KUKA KRL program: EPS_2_251825_SA24_A_20260116064100.src

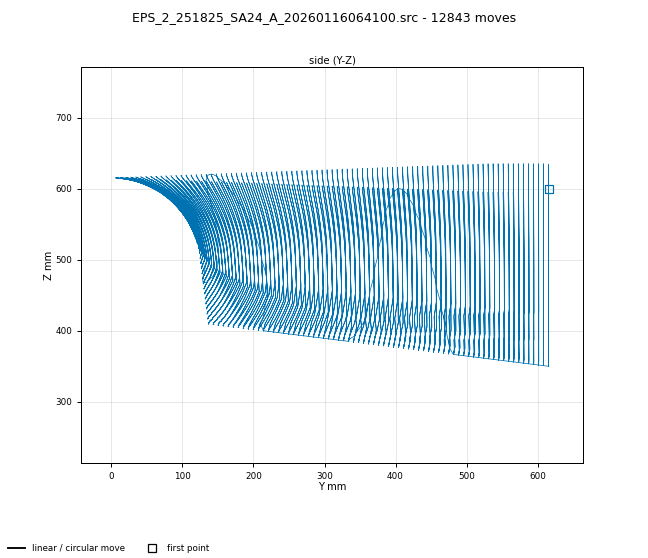
[picture p0: tool path of EPS_2_251825_SA24_A_20260116064100.src, 12843 of 12845 moves have a stored position in this frame; points joined in program order, loops and branches not executed]
&ACCESS RVP
&REL 4
&COMMENT QRS 19112012
&PARAM EDITMASK = *
DEF PART()
EXT BAS (BAS_COMMAND :IN,REAL :IN )
INT I
BAS (#INITMOV,0 )

;KUKA QRS Post kuka4.cps  Date:22-06-2017 !

File_ID=2983

QRS_PRE_INIT()

;Init var - Until changes are made in qrs_pre_init
Outlet_Square_prg=0
Inlet_1_Square_prg=0
Inlet_2_Square_prg=0
Inlet_3_Square_prg=0
Inlet_4_Square_prg=0
Inlet_5_Square_prg=0

Outlet_1={X 0.000, Y 530.070, Z 534.500, B 0.000, E1 0.000 }
Inlet_1={X 0.000, Y 532.930, Z 494.500, B 0.000, E1 180.000 }
Outlet_1_type=201
Inlet_1_type=201
;QRS#1=Sidecore dimensions
;QRS#2=200-8" PVC SDR 35
;QRS#3=200-8" PVC SDR 35
;QRS#4=
;QRS#5=
;QRS#6=
;QRS#7=
;QRS#8=
;QRS#9=12-08 PSX
;QRS#10=12-08 PSX
;QRS#11=
;QRS#12=
;QRS#13=
;QRS#14=
;QRS#15=
;QRS#16=1220x127x914 3'
;QRS#17=EPS Height
;QRS#18=635
;QRS#19=*
;QRS#20= UPDATED VERSION 22-06-2017
;QRS#21=*
Outlet_Square=0100
Inlet_1_Square=0100
Inlet_2_Square=0
Inlet_3_Square=0
Inlet_4_Square=0
Inlet_5_Square=0
Mill_Square=1
Outlet_Square_Prg=204
Inlet_1_Square_prg=204

QRS_INIT()

$ADVANCE=5

; T1
PTP {E1 173.589,E2 173.589}
PTP {X 0,Y 615.513,A -85,B 0,C 180,E1 173.589,E2 173.589,E3 0,E4 0,E5 0,E6 0}
QRS_SPEED_INIT()
LIN {X 0,Y 615.513,Z 600,A -85,B 0,C 180,E1 173.589,E2 173.589,E3 0,E4 0,E5 0,E6 0} C_VEL
LIN {X 0,Y 615.513,Z 359.866,A -85,B 0,C 180,E1 173.589,E2 173.589} C_VEL
LIN {X 0,Y 615.513,Z 351.692,A -85,B 0,C 180,E1 173.589,E2 173.589} C_VEL
LIN {X 0,Y 615.497,Z 349.692,A -85,B 0,C 180,E1 173.403,E2 173.403} C_VEL
LIN {X 0,Y 615.488,Z 349.69,A -85,B 0,C 180,E1 170.801,E2 170.801} C_VEL
LIN {X 0,Y 615.478,Z 349.685,A -85,B 0,C 180,E1 168.139,E2 168.139} C_VEL
LIN {X 0,Y 615.497,Z 349.694,A -85,B 0,C 180,E1 165.451,E2 165.451} C_VEL
LIN {X 0,Y 615.493,Z 349.685,A -85,B 0,C 180,E1 162.73,E2 162.73} C_VEL
LIN {X 0,Y 615.479,Z 349.687,A -85,B 0,C 180,E1 159.967,E2 159.967} C_VEL
LIN {X 0,Y 615.488,Z 349.695,A -85,B 0,C 180,E1 157.155,E2 157.155} C_VEL
LIN {X 0,Y 615.484,Z 349.683,A -85,B 0,C 180,E1 154.429,E2 154.429} C_VEL
LIN {X 0,Y 615.497,Z 349.697,A -85,B 0,C 180,E1 151.546,E2 151.546} C_VEL
LIN {X 0,Y 615.487,Z 349.686,A -85,B 0,C 180,E1 148.912,E2 148.912} C_VEL
LIN {X 0,Y 615.484,Z 349.683,A -85,B 0,C 180,E1 146.464,E2 146.464} C_VEL
LIN {X 0,Y 615.488,Z 349.702,A -85,B 0,C 180,E1 143.575,E2 143.575} C_VEL
LIN {X 0,Y 615.481,Z 349.686,A -85,B 0,C 180,E1 140.937,E2 140.937} C_VEL
LIN {X 0,Y 615.485,Z 349.683,A -85,B 0,C 180,E1 138.526,E2 138.526} C_VEL
LIN {X 0,Y 615.491,Z 349.695,A -85,B 0,C 180,E1 135.85,E2 135.85} C_VEL
LIN {X 0,Y 615.483,Z 349.686,A -85,B 0,C 180,E1 133.047,E2 133.047} C_VEL
LIN {X 0,Y 615.482,Z 349.684,A -85,B 0,C 180,E1 130.606,E2 130.606} C_VEL
LIN {X 0,Y 615.484,Z 349.695,A -85,B 0,C 180,E1 128.011,E2 128.011} C_VEL
LIN {X 0,Y 615.486,Z 349.696,A -85,B 0,C 180,E1 125.615,E2 125.615} C_VEL
LIN {X 0,Y 615.477,Z 349.688,A -85,B 0,C 180,E1 123.236,E2 123.236} C_VEL
LIN {X 0,Y 615.492,Z 349.681,A -85,B 0,C 180,E1 120.919,E2 120.919} C_VEL
LIN {X 0,Y 615.477,Z 349.689,A -85,B 0,C 180,E1 118.448,E2 118.448} C_VEL
LIN {X 0,Y 615.489,Z 349.695,A -85,B 0,C 180,E1 115.715,E2 115.715} C_VEL
LIN {X 0,Y 615.486,Z 349.683,A -85,B 0,C 180,E1 112.844,E2 112.844} C_VEL
LIN {X 0,Y 615.485,Z 349.703,A -85,B 0,C 180,E1 110.032,E2 110.032} C_VEL
LIN {X 0,Y 615.481,Z 349.809,A -85,B 0,C 180,E1 108.602,E2 108.602} C_VEL
LIN {X 0,Y 615.486,Z 366.721,A -85,B 0,C 180,E1 105.735,E2 105.735} C_VEL
LIN {X 0,Y 615.497,Z 384.117,A -85,B 0,C 180,E1 102.823,E2 102.823} C_VEL
LIN {X 0,Y 615.478,Z 491.809,A -85,B 0,C 180,E1 101.527,E2 101.527} C_VEL
LIN {X 0,Y 615.481,Z 504.75,A -85,B 0,C 180,E1 101.235,E2 101.235} C_VEL
LIN {X 0,Y 615.493,Z 516.589,A -85,B 0,C 180,E1 100.843,E2 100.843} C_VEL
LIN {X 0,Y 615.485,Z 527.572,A -85,B 0,C 180,E1 100.36,E2 100.36} C_VEL
LIN {X 0,Y 615.492,Z 539.308,A -85,B 0,C 180,E1 99.696,E2 99.696} C_VEL
LIN {X 0,Y 615.499,Z 549.77,A -85,B 0,C 180,E1 98.95,E2 98.95} C_VEL
LIN {X 0,Y 615.498,Z 558.332,A -85,B 0,C 180,E1 98.206,E2 98.206} C_VEL
LIN {X 0,Y 615.497,Z 566.211,A -85,B 0,C 180,E1 97.38,E2 97.38} C_VEL
LIN {X 0,Y 615.497,Z 573.9,A -85,B 0,C 180,E1 96.392,E2 96.392} C_VEL
LIN {X 0,Y 615.497,Z 580.959,A -85,B 0,C 180,E1 95.241,E2 95.241} C_VEL
LIN {X 0,Y 615.494,Z 585.658,A -85,B 0,C 180,E1 94.256,E2 94.256} C_VEL
LIN {X 0,Y 615.494,Z 589.255,A -85,B 0,C 180,E1 93.273,E2 93.273} C_VEL
LIN {X 0,Y 615.496,Z 591.115,A -85,B 0,C 180,E1 92.618,E2 92.618} C_VEL
LIN {X 0,Y 615.499,Z 592.533,A -85,B 0,C 180,E1 91.963,E2 91.963} C_VEL
LIN {X 0,Y 615.496,Z 594.142,A -85,B 0,C 180,E1 90.654,E2 90.654} C_VEL
LIN {X 0,Y 615.495,Z 594.384,A -85,B 0,C 180,E1 90,E2 90} C_VEL
LIN {X 0,Y 615.495,Z 594.206,A -85,B 0,C 180,E1 89.346,E2 89.346} C_VEL
LIN {X 0,Y 615.499,Z 592.682,A -85,B 0,C 180,E1 88.037,E2 88.037} C_VEL
LIN {X 0,Y 615.498,Z 591.341,A -85,B 0,C 180,E1 87.382,E2 87.382} C_VEL
LIN {X 0,Y 615.496,Z 588.494,A -85,B 0,C 180,E1 86.399,E2 86.399} C_VEL
LIN {X 0,Y 615.499,Z 584.635,A -85,B 0,C 180,E1 85.416,E2 85.416} C_VEL
LIN {X 0,Y 615.498,Z 579.652,A -85,B 0,C 180,E1 84.43,E2 84.43} C_VEL
LIN {X 0,Y 615.496,Z 573.208,A -85,B 0,C 180,E1 83.418,E2 83.418} C_VEL
LIN {X 0,Y 615.497,Z 565.538,A -85,B 0,C 180,E1 82.455,E2 82.455} C_VEL
LIN {X 0,Y 615.498,Z 555.761,A -85,B 0,C 180,E1 81.464,E2 81.464} C_VEL
LIN {X 0,Y 615.498,Z 545.496,A -85,B 0,C 180,E1 80.636,E2 80.636} C_VEL
LIN {X 0,Y 615.488,Z 533.934,A -85,B 0,C 180,E1 79.889,E2 79.889} C_VEL
LIN {X 0,Y 615.495,Z 522.053,A -85,B 0,C 180,E1 79.292,E2 79.292} C_VEL
LIN {X 0,Y 615.483,Z 509.169,A -85,B 0,C 180,E1 78.807,E2 78.807} C_VEL
LIN {X 0,Y 615.476,Z 496.573,A -85,B 0,C 180,E1 78.473,E2 78.473} C_VEL
LIN {X 0,Y 615.48,Z 483.461,A -85,B 0,C 180,E1 78.265,E2 78.265} C_VEL
LIN {X 0,Y 615.499,Z 384.153,A -85,B 0,C 180,E1 77.093,E2 77.093} C_VEL
LIN {X 0,Y 615.486,Z 367.257,A -85,B 0,C 180,E1 74.265,E2 74.265} C_VEL
LIN {X 0,Y 615.487,Z 350.325,A -85,B 0,C 180,E1 71.396,E2 71.396} C_VEL
LIN {X 0,Y 615.491,Z 349.685,A -85,B 0,C 180,E1 71.268,E2 71.268} C_VEL
LIN {X 0,Y 615.477,Z 349.687,A -85,B 0,C 180,E1 68.568,E2 68.568} C_VEL
LIN {X 0,Y 615.482,Z 349.696,A -85,B 0,C 180,E1 65.728,E2 65.728} C_VEL
LIN {X 0,Y 615.486,Z 349.683,A -85,B 0,C 180,E1 62.956,E2 62.956} C_VEL
LIN {X 0,Y 615.497,Z 349.695,A -85,B 0,C 180,E1 60.204,E2 60.204} C_VEL
LIN {X 0,Y 615.48,Z 349.688,A -85,B 0,C 180,E1 57.543,E2 57.543} C_VEL
LIN {X 0,Y 615.499,Z 349.68,A -85,B 0,C 180,E1 55.187,E2 55.187} C_VEL
LIN {X 0,Y 615.477,Z 349.688,A -85,B 0,C 180,E1 52.758,E2 52.758} C_VEL
LIN {X 0,Y 615.48,Z 349.695,A -85,B 0,C 180,E1 49.912,E2 49.912} C_VEL
LIN {X 0,Y 615.475,Z 349.689,A -85,B 0,C 180,E1 47.647,E2 47.647} C_VEL
LIN {X 0,Y 615.48,Z 349.686,A -85,B 0,C 180,E1 44.932,E2 44.932} C_VEL
LIN {X 0,Y 615.486,Z 349.695,A -85,B 0,C 180,E1 42.082,E2 42.082} C_VEL
LIN {X 0,Y 615.477,Z 349.688,A -85,B 0,C 180,E1 39.751,E2 39.751} C_VEL
LIN {X 0,Y 615.478,Z 349.688,A -85,B 0,C 180,E1 36.937,E2 36.937} C_VEL
LIN {X 0,Y 615.481,Z 349.692,A -85,B 0,C 180,E1 34.023,E2 34.023} C_VEL
LIN {X 0,Y 615.479,Z 349.686,A -85,B 0,C 180,E1 31.686,E2 31.686} C_VEL
LIN {X 0,Y 615.486,Z 349.683,A -85,B 0,C 180,E1 29.407,E2 29.407} C_VEL
LIN {X 0,Y 615.495,Z 349.698,A -85,B 0,C 180,E1 26.444,E2 26.444} C_VEL
LIN {X 0,Y 615.486,Z 349.683,A -85,B 0,C 180,E1 23.557,E2 23.557} C_VEL
LIN {X 0,Y 615.486,Z 349.698,A -85,B 0,C 180,E1 20.731,E2 20.731} C_VEL
LIN {X 0,Y 615.477,Z 349.687,A -85,B 0,C 180,E1 17.957,E2 17.957} C_VEL
LIN {X 0,Y 615.491,Z 349.686,A -85,B 0,C 180,E1 15.226,E2 15.226} C_VEL
LIN {X 0,Y 615.493,Z 349.695,A -85,B 0,C 180,E1 12.53,E2 12.53} C_VEL
LIN {X 0,Y 615.477,Z 349.685,A -85,B 0,C 180,E1 9.862,E2 9.862} C_VEL
LIN {X 0,Y 615.49,Z 349.689,A -85,B 0,C 180,E1 7.216,E2 7.216} C_VEL
LIN {X 0,Y 615.494,Z 349.693,A -85,B 0,C 180,E1 4.585,E2 4.585} C_VEL
LIN {X 0,Y 615.477,Z 349.685,A -85,B 0,C 180,E1 1.963,E2 1.963} C_VEL
LIN {X 0,Y 615.489,Z 349.688,A -85,B 0,C 180,E1 -0.654,E2 -0.654} C_VEL
LIN {X 0,Y 615.496,Z 349.693,A -85,B 0,C 180,E1 -3.273,E2 -3.273} C_VEL
LIN {X 0,Y 615.476,Z 349.685,A -85,B 0,C 180,E1 -5.899,E2 -5.899} C_VEL
LIN {X 0,Y 615.491,Z 349.688,A -85,B 0,C 180,E1 -8.537,E2 -8.537} C_VEL
LIN {X 0,Y 615.494,Z 349.692,A -85,B 0,C 180,E1 -11.193,E2 -11.193} C_VEL
LIN {X 0,Y 615.474,Z 349.685,A -85,B 0,C 180,E1 -13.933,E2 -13.933} C_VEL
LIN {X 0,Y 615.493,Z 349.692,A -85,B 0,C 180,E1 -16.587,E2 -16.587} C_VEL
LIN {X 0,Y 615.49,Z 349.687,A -85,B 0,C 180,E1 -19.338,E2 -19.338} C_VEL
LIN {X 0,Y 615.479,Z 349.687,A -85,B 0,C 180,E1 -22.137,E2 -22.137} C_VEL
LIN {X 0,Y 615.488,Z 349.694,A -85,B 0,C 180,E1 -24.992,E2 -24.992} C_VEL
LIN {X 0,Y 615.487,Z 349.688,A -85,B 0,C 180,E1 -27.177,E2 -27.177} C_VEL
LIN {X 0,Y 615.477,Z 349.685,A -85,B 0,C 180,E1 -29.795,E2 -29.795} C_VEL
LIN {X 0,Y 615.495,Z 349.694,A -85,B 0,C 180,E1 -32.457,E2 -32.457} C_VEL
LIN {X 0,Y 615.49,Z 349.695,A -85,B 0,C 180,E1 -34.815,E2 -34.815} C_VEL
LIN {X 0,Y 615.491,Z 349.684,A -85,B 0,C 180,E1 -37.242,E2 -37.242} C_VEL
LIN {X 0,Y 615.484,Z 349.69,A -85,B 0,C 180,E1 -40.09,E2 -40.09} C_VEL
LIN {X 0,Y 615.499,Z 349.695,A -85,B 0,C 180,E1 -42.352,E2 -42.352} C_VEL
LIN {X 0,Y 615.484,Z 349.686,A -85,B 0,C 180,E1 -45.069,E2 -45.069} C_VEL
LIN {X 0,Y 615.477,Z 349.69,A -85,B 0,C 180,E1 -47.921,E2 -47.921} C_VEL
LIN {X 0,Y 615.497,Z 349.696,A -85,B 0,C 180,E1 -50.252,E2 -50.252} C_VEL
LIN {X 0,Y 615.485,Z 349.685,A -85,B 0,C 180,E1 -53.064,E2 -53.064} C_VEL
LIN {X 0,Y 615.491,Z 349.681,A -85,B 0,C 180,E1 -55.299,E2 -55.299} C_VEL
LIN {X 0,Y 615.477,Z 349.688,A -85,B 0,C 180,E1 -57.671,E2 -57.671} C_VEL
LIN {X 0,Y 615.499,Z 349.699,A -85,B 0,C 180,E1 -60.204,E2 -60.204} C_VEL
LIN {X 0,Y 615.487,Z 349.684,A -85,B 0,C 180,E1 -62.956,E2 -62.956} C_VEL
LIN {X 0,Y 615.478,Z 349.691,A -85,B 0,C 180,E1 -65.728,E2 -65.728} C_VEL
LIN {X 0,Y 615.48,Z 349.76,A -85,B 0,C 180,E1 -67.438,E2 -67.438} C_VEL
LIN {X 0,Y 615.494,Z 369.694,A -85,B 0,C 180,E1 -70.142,E2 -70.142} C_VEL
LIN {X 0,Y 615.493,Z 391.661,A -85,B 0,C 180,E1 -73.072,E2 -73.072} C_VEL
LIN {X 0,Y 615.498,Z 414.417,A -85,B 0,C 180,E1 -76.064,E2 -76.064} C_VEL
LIN {X 0,Y 615.497,Z 422.467,A -85,B 0,C 180,E1 -77.114,E2 -77.114} C_VEL
LIN {X 0,Y 615.479,Z 530.847,A -85,B 0,C 180,E1 -78.411,E2 -78.411} C_VEL
LIN {X 0,Y 615.478,Z 543.355,A -85,B 0,C 180,E1 -78.682,E2 -78.682} C_VEL
LIN {X 0,Y 615.491,Z 556.569,A -85,B 0,C 180,E1 -79.111,E2 -79.111} C_VEL
LIN {X 0,Y 615.478,Z 568.483,A -85,B 0,C 180,E1 -79.639,E2 -79.639} C_VEL
LIN {X 0,Y 615.487,Z 579.999,A -85,B 0,C 180,E1 -80.304,E2 -80.304} C_VEL
LIN {X 0,Y 615.499,Z 590.344,A -85,B 0,C 180,E1 -81.05,E2 -81.05} C_VEL
LIN {X 0,Y 615.497,Z 598.814,A -85,B 0,C 180,E1 -81.794,E2 -81.794} C_VEL
LIN {X 0,Y 615.498,Z 606.608,A -85,B 0,C 180,E1 -82.62,E2 -82.62} C_VEL
LIN {X 0,Y 615.496,Z 614.204,A -85,B 0,C 180,E1 -83.608,E2 -83.608} C_VEL
LIN {X 0,Y 615.498,Z 621.205,A -85,B 0,C 180,E1 -84.759,E2 -84.759} C_VEL
LIN {X 0,Y 615.493,Z 625.852,A -85,B 0,C 180,E1 -85.744,E2 -85.744} C_VEL
LIN {X 0,Y 615.495,Z 629.399,A -85,B 0,C 180,E1 -86.727,E2 -86.727} C_VEL
LIN {X 0,Y 615.497,Z 631.233,A -85,B 0,C 180,E1 -87.382,E2 -87.382} C_VEL
LIN {X 0,Y 615.497,Z 632.608,A -85,B 0,C 180,E1 -88.037,E2 -88.037} C_VEL
LIN {X 0,Y 615.496,Z 634.174,A -85,B 0,C 180,E1 -89.346,E2 -89.346} C_VEL
LIN {X 0,Y 615.494,Z 634.389,A -85,B 0,C 180,E1 -90,E2 -90} C_VEL
LIN {X 0,Y 615.496,Z 633.58,A -85,B 0,C 180,E1 -91.309,E2 -91.309} C_VEL
LIN {X 0,Y 615.497,Z 632.608,A -85,B 0,C 180,E1 -91.963,E2 -91.963} C_VEL
LIN {X 0,Y 615.497,Z 631.233,A -85,B 0,C 180,E1 -92.618,E2 -92.618} C_VEL
LIN {X 0,Y 615.496,Z 628.35,A -85,B 0,C 180,E1 -93.601,E2 -93.601} C_VEL
LIN {X 0,Y 615.498,Z 624.442,A -85,B 0,C 180,E1 -94.584,E2 -94.584} C_VEL
LIN {X 0,Y 615.499,Z 619.406,A -85,B 0,C 180,E1 -95.57,E2 -95.57} C_VEL
LIN {X 0,Y 615.497,Z 612.869,A -85,B 0,C 180,E1 -96.583,E2 -96.583} C_VEL
LIN {X 0,Y 615.497,Z 605.135,A -85,B 0,C 180,E1 -97.545,E2 -97.545} C_VEL
LIN {X 0,Y 615.498,Z 597.047,A -85,B 0,C 180,E1 -98.371,E2 -98.371} C_VEL
LIN {X 0,Y 615.499,Z 587.17,A -85,B 0,C 180,E1 -99.198,E2 -99.198} C_VEL
LIN {X 0,Y 615.488,Z 575.985,A -85,B 0,C 180,E1 -99.945,E2 -99.945} C_VEL
LIN {X 0,Y 615.481,Z 565.029,A -85,B 0,C 180,E1 -100.527,E2 -100.527} C_VEL
LIN {X 0,Y 615.49,Z 552.453,A -85,B 0,C 180,E1 -101.041,E2 -101.041} C_VEL
LIN {X 0,Y 615.477,Z 540.079,A -85,B 0,C 180,E1 -101.401,E2 -101.401} C_VEL
LIN {X 0,Y 615.481,Z 526.487,A -85,B 0,C 180,E1 -101.652,E2 -101.652} C_VEL
LIN {X 0,Y 615.497,Z 422.467,A -85,B 0,C 180,E1 -102.886,E2 -102.886} C_VEL
LIN {X 0,Y 615.49,Z 399.409,A -85,B 0,C 180,E1 -105.905,E2 -105.905} C_VEL
LIN {X 0,Y 615.494,Z 377.451,A -85,B 0,C 180,E1 -108.818,E2 -108.818} C_VEL
LIN {X 0,Y 615.483,Z 356.76,A -85,B 0,C 180,E1 -111.607,E2 -111.607} C_VEL
LIN {X 0,Y 615.481,Z 349.685,A -85,B 0,C 180,E1 -112.593,E2 -112.593} C_VEL
LIN {X 0,Y 615.488,Z 349.683,A -85,B 0,C 180,E1 -114.991,E2 -114.991} C_VEL
LIN {X 0,Y 615.487,Z 349.698,A -85,B 0,C 180,E1 -117.914,E2 -117.914} C_VEL
LIN {X 0,Y 615.476,Z 349.692,A -85,B 0,C 180,E1 -120.16,E2 -120.16} C_VEL
LIN {X 0,Y 615.479,Z 349.686,A -85,B 0,C 180,E1 -122.457,E2 -122.457} C_VEL
LIN {X 0,Y 615.499,Z 349.68,A -85,B 0,C 180,E1 -124.813,E2 -124.813} C_VEL
LIN {X 0,Y 615.483,Z 349.69,A -85,B 0,C 180,E1 -127.241,E2 -127.241} C_VEL
LIN {X 0,Y 615.477,Z 349.691,A -85,B 0,C 180,E1 -130.088,E2 -130.088} C_VEL
LIN {X 0,Y 615.475,Z 349.686,A -85,B 0,C 180,E1 -132.353,E2 -132.353} C_VEL
LIN {X 0,Y 615.486,Z 349.688,A -85,B 0,C 180,E1 -135.067,E2 -135.067} C_VEL
LIN {X 0,Y 615.486,Z 349.69,A -85,B 0,C 180,E1 -137.918,E2 -137.918} C_VEL
LIN {X 0,Y 615.477,Z 349.686,A -85,B 0,C 180,E1 -140.249,E2 -140.249} C_VEL
LIN {X 0,Y 615.488,Z 349.69,A -85,B 0,C 180,E1 -143.062,E2 -143.062} C_VEL
LIN {X 0,Y 615.481,Z 349.688,A -85,B 0,C 180,E1 -145.978,E2 -145.978} C_VEL
LIN {X 0,Y 615.476,Z 349.685,A -85,B 0,C 180,E1 -148.314,E2 -148.314} C_VEL
LIN {X 0,Y 615.488,Z 349.684,A -85,B 0,C 180,E1 -150.594,E2 -150.594} C_VEL
LIN {X 0,Y 615.497,Z 349.691,A -85,B 0,C 180,E1 -153.556,E2 -153.556} C_VEL
LIN {X 0,Y 615.486,Z 349.683,A -85,B 0,C 180,E1 -156.444,E2 -156.444} C_VEL
LIN {X 0,Y 615.497,Z 349.699,A -85,B 0,C 180,E1 -159.27,E2 -159.27} C_VEL
LIN {X 0,Y 615.477,Z 349.685,A -85,B 0,C 180,E1 -162.043,E2 -162.043} C_VEL
LIN {X 0,Y 615.492,Z 349.69,A -85,B 0,C 180,E1 -164.774,E2 -164.774} C_VEL
LIN {X 0,Y 615.491,Z 349.69,A -85,B 0,C 180,E1 -167.47,E2 -167.47} C_VEL
LIN {X 0,Y 615.477,Z 349.685,A -85,B 0,C 180,E1 -170.138,E2 -170.138} C_VEL
LIN {X 0,Y 615.494,Z 349.692,A -85,B 0,C 180,E1 -172.784,E2 -172.784} C_VEL
LIN {X 0,Y 615.492,Z 349.689,A -85,B 0,C 180,E1 -175.415,E2 -175.415} C_VEL
LIN {X 0,Y 615.477,Z 349.685,A -85,B 0,C 180,E1 -178.037,E2 -178.037} C_VEL
LIN {X 0,Y 615.494,Z 349.692,A -85,B 0,C 180,E1 -180.654,E2 -180.654} C_VEL
LIN {X 0,Y 615.492,Z 349.689,A -85,B 0,C 180,E1 -183.273,E2 -183.273} C_VEL
LIN {X 0,Y 615.476,Z 349.685,A -85,B 0,C 180,E1 -185.899,E2 -185.899} C_VEL
LIN {X 0,Y 615.497,Z 349.692,A -85,B 0,C 180,E1 -186.597,E2 -186.597} C_VEL
LIN {X 0,Y 614.817,Z 349.838,A -85,B 0,C 180,E1 -187.143,E2 -187.143} C_VEL
LIN {X 0,Y 611.977,Z 350.249,A -85,B 0,C 180,E1 -188.029,E2 -188.029} C_VEL
LIN {X 0,Y 609.583,Z 350.561,A -85,B 0,C 180,E1 -188.741,E2 -188.741} C_VEL
LIN {X 0,Y 608.546,Z 350.679,A -85,B 0,C 180,E1 -189.291,E2 -189.291} C_VEL
LIN {X 0,Y 608.456,Z 350.688,A -85,B 0,C 180,E1 -189.477,E2 -189.477} C_VEL
LIN {X 0,Y 608.456,Z 350.687,A -85,B 0,C 180,E1 -192,E2 -192} C_VEL
LIN {X 0,Y 608.481,Z 350.694,A -85,B 0,C 180,E1 -194.72,E2 -194.72} C_VEL
LIN {X 0,Y 608.453,Z 350.688,A -85,B 0,C 180,E1 -197.477,E2 -197.477} C_VEL
LIN {X 0,Y 608.462,Z 350.69,A -85,B 0,C 180,E1 -200.274,E2 -200.274} C_VEL
LIN {X 0,Y 608.486,Z 350.691,A -85,B 0,C 180,E1 -202.485,E2 -202.485} C_VEL
LIN {X 0,Y 608.449,Z 350.689,A -85,B 0,C 180,E1 -205.301,E2 -205.301} C_VEL
LIN {X 0,Y 608.444,Z 350.688,A -85,B 0,C 180,E1 -207.518,E2 -207.518} C_VEL
LIN {X 0,Y 608.46,Z 350.688,A -85,B 0,C 180,E1 -209.973,E2 -209.973} C_VEL
LIN {X 0,Y 608.467,Z 350.696,A -85,B 0,C 180,E1 -212.525,E2 -212.525} C_VEL
LIN {X 0,Y 608.436,Z 350.69,A -85,B 0,C 180,E1 -215.278,E2 -215.278} C_VEL
LIN {X 0,Y 608.467,Z 350.687,A -85,B 0,C 180,E1 -217.747,E2 -217.747} C_VEL
LIN {X 0,Y 608.449,Z 350.698,A -85,B 0,C 180,E1 -220.33,E2 -220.33} C_VEL
LIN {X 0,Y 608.483,Z 350.684,A -85,B 0,C 180,E1 -223.312,E2 -223.312} C_VEL
LIN {X 0,Y 608.467,Z 350.693,A -85,B 0,C 180,E1 -226.132,E2 -226.132} C_VEL
LIN {X 0,Y 608.451,Z 350.69,A -85,B 0,C 180,E1 -228.824,E2 -228.824} C_VEL
LIN {X 0,Y 608.468,Z 350.686,A -85,B 0,C 180,E1 -231.413,E2 -231.413} C_VEL
LIN {X 0,Y 608.476,Z 350.691,A -85,B 0,C 180,E1 -233.951,E2 -233.951} C_VEL
LIN {X 0,Y 608.448,Z 350.696,A -85,B 0,C 180,E1 -236.329,E2 -236.329} C_VEL
LIN {X 0,Y 608.476,Z 350.686,A -85,B 0,C 180,E1 -238.728,E2 -238.728} C_VEL
LIN {X 0,Y 608.469,Z 350.686,A -85,B 0,C 180,E1 -241.381,E2 -241.381} C_VEL
LIN {X 0,Y 608.471,Z 350.692,A -85,B 0,C 180,E1 -244.28,E2 -244.28} C_VEL
LIN {X 0,Y 608.449,Z 350.688,A -85,B 0,C 180,E1 -246.877,E2 -246.877} C_VEL
LIN {X 0,Y 608.459,Z 350.693,A -85,B 0,C 180,E1 -249.726,E2 -249.726} C_VEL
LIN {X 0,Y 608.467,Z 350.778,A -85,B 0,C 180,E1 -251.331,E2 -251.331} C_VEL
LIN {X 0,Y 608.497,Z 366.845,A -85,B 0,C 180,E1 -254.08,E2 -254.08} C_VEL
LIN {X 0,Y 608.485,Z 384.321,A -85,B 0,C 180,E1 -257.027,E2 -257.027} C_VEL
LIN {X 0,Y 608.573,Z 393.682,A -85,B 0,C 180,E1 -257.156,E2 -257.156} C_VEL
LIN {X 0,Y 608.545,Z 490.809,A -85,B 0,C 180,E1 -258.319,E2 -258.319} C_VEL
LIN {X 0,Y 608.524,Z 504.124,A -85,B 0,C 180,E1 -258.614,E2 -258.614} C_VEL
LIN {X 0,Y 608.527,Z 517.379,A -85,B 0,C 180,E1 -259.056,E2 -259.056} C_VEL
LIN {X 0,Y 608.495,Z 529.373,A -85,B 0,C 180,E1 -259.603,E2 -259.603} C_VEL
LIN {X 0,Y 608.505,Z 540.793,A -85,B 0,C 180,E1 -260.276,E2 -260.276} C_VEL
LIN {X 0,Y 608.474,Z 551.086,A -85,B 0,C 180,E1 -261.03,E2 -261.03} C_VEL
LIN {X 0,Y 608.464,Z 560.352,A -85,B 0,C 180,E1 -261.866,E2 -261.866} C_VEL
LIN {X 0,Y 608.466,Z 569.325,A -85,B 0,C 180,E1 -262.868,E2 -262.868} C_VEL
LIN {X 0,Y 608.444,Z 576.556,A -85,B 0,C 180,E1 -263.867,E2 -263.867} C_VEL
LIN {X 0,Y 608.462,Z 581.435,A -85,B 0,C 180,E1 -264.698,E2 -264.698} C_VEL
LIN {X 0,Y 608.439,Z 586.179,A -85,B 0,C 180,E1 -265.694,E2 -265.694} C_VEL
LIN {X 0,Y 608.425,Z 589.812,A -85,B 0,C 180,E1 -266.689,E2 -266.689} C_VEL
LIN {X 0,Y 608.425,Z 591.691,A -85,B 0,C 180,E1 -267.352,E2 -267.352} C_VEL
LIN {X 0,Y 608.444,Z 593.127,A -85,B 0,C 180,E1 -268.014,E2 -268.014} C_VEL
LIN {X 0,Y 608.439,Z 594.752,A -85,B 0,C 180,E1 -269.338,E2 -269.338} C_VEL
LIN {X 0,Y 608.435,Z 594.995,A -85,B 0,C 180,E1 -270,E2 -270} C_VEL
LIN {X 0,Y 608.438,Z 594.815,A -85,B 0,C 180,E1 -270.662,E2 -270.662} C_VEL
LIN {X 0,Y 608.444,Z 593.276,A -85,B 0,C 180,E1 -271.986,E2 -271.986} C_VEL
LIN {X 0,Y 608.426,Z 591.919,A -85,B 0,C 180,E1 -272.648,E2 -272.648} C_VEL
LIN {X 0,Y 608.449,Z 589.042,A -85,B 0,C 180,E1 -273.642,E2 -273.642} C_VEL
LIN {X 0,Y 608.433,Z 585.143,A -85,B 0,C 180,E1 -274.638,E2 -274.638} C_VEL
LIN {X 0,Y 608.45,Z 580.113,A -85,B 0,C 180,E1 -275.634,E2 -275.634} C_VEL
LIN {X 0,Y 608.441,Z 573.796,A -85,B 0,C 180,E1 -276.633,E2 -276.633} C_VEL
LIN {X 0,Y 608.475,Z 565.88,A -85,B 0,C 180,E1 -277.633,E2 -277.633} C_VEL
LIN {X 0,Y 608.472,Z 556.038,A -85,B 0,C 180,E1 -278.636,E2 -278.636} C_VEL
LIN {X 0,Y 608.48,Z 545.717,A -85,B 0,C 180,E1 -279.473,E2 -279.473} C_VEL
LIN {X 0,Y 608.485,Z 534.104,A -85,B 0,C 180,E1 -280.229,E2 -280.229} C_VEL
LIN {X 0,Y 608.526,Z 522.887,A -85,B 0,C 180,E1 -280.802,E2 -280.802} C_VEL
LIN {X 0,Y 608.523,Z 510.37,A -85,B 0,C 180,E1 -281.287,E2 -281.287} C_VEL
LIN {X 0,Y 608.521,Z 497.571,A -85,B 0,C 180,E1 -281.639,E2 -281.639} C_VEL
LIN {X 0,Y 608.534,Z 485.31,A -85,B 0,C 180,E1 -281.85,E2 -281.85} C_VEL
LIN {X 0,Y 608.463,Z 384.352,A -85,B 0,C 180,E1 -283.059,E2 -283.059} C_VEL
LIN {X 0,Y 608.497,Z 367.375,A -85,B 0,C 180,E1 -285.92,E2 -285.92} C_VEL
LIN {X 0,Y 608.471,Z 350.687,A -85,B 0,C 180,E1 -288.775,E2 -288.775} C_VEL
LIN {X 0,Y 608.467,Z 350.69,A -85,B 0,C 180,E1 -291.691,E2 -291.691} C_VEL
LIN {X 0,Y 608.452,Z 350.69,A -85,B 0,C 180,E1 -294.57,E2 -294.57} C_VEL
LIN {X 0,Y 608.476,Z 350.685,A -85,B 0,C 180,E1 -297.206,E2 -297.206} C_VEL
LIN {X 0,Y 608.47,Z 350.696,A -85,B 0,C 180,E1 -299.971,E2 -299.971} C_VEL
LIN {X 0,Y 608.456,Z 350.689,A -85,B 0,C 180,E1 -302.521,E2 -302.521} C_VEL
LIN {X 0,Y 608.447,Z 350.69,A -85,B 0,C 180,E1 -305.276,E2 -305.276} C_VEL
LIN {X 0,Y 608.466,Z 350.695,A -85,B 0,C 180,E1 -307.745,E2 -307.745} C_VEL
LIN {X 0,Y 608.446,Z 350.691,A -85,B 0,C 180,E1 -310.328,E2 -310.328} C_VEL
LIN {X 0,Y 608.447,Z 350.688,A -85,B 0,C 180,E1 -312.959,E2 -312.959} C_VEL
LIN {X 0,Y 608.458,Z 350.698,A -85,B 0,C 180,E1 -315.735,E2 -315.735} C_VEL
LIN {X 0,Y 608.459,Z 350.686,A -85,B 0,C 180,E1 -318.657,E2 -318.657} C_VEL
LIN {X 0,Y 608.464,Z 350.692,A -85,B 0,C 180,E1 -321.411,E2 -321.411} C_VEL
LIN {X 0,Y 608.471,Z 350.69,A -85,B 0,C 180,E1 -323.95,E2 -323.95} C_VEL
LIN {X 0,Y 608.461,Z 350.687,A -85,B 0,C 180,E1 -326.329,E2 -326.329} C_VEL
LIN {X 0,Y 608.472,Z 350.685,A -85,B 0,C 180,E1 -328.726,E2 -328.726} C_VEL
LIN {X 0,Y 608.475,Z 350.693,A -85,B 0,C 180,E1 -331.377,E2 -331.377} C_VEL
LIN {X 0,Y 608.464,Z 350.686,A -85,B 0,C 180,E1 -334.278,E2 -334.278} C_VEL
LIN {X 0,Y 608.449,Z 350.69,A -85,B 0,C 180,E1 -336.876,E2 -336.876} C_VEL
LIN {X 0,Y 608.469,Z 350.695,A -85,B 0,C 180,E1 -339.318,E2 -339.318} C_VEL
LIN {X 0,Y 608.446,Z 350.691,A -85,B 0,C 180,E1 -341.828,E2 -341.828} C_VEL
LIN {X 0,Y 608.47,Z 350.686,A -85,B 0,C 180,E1 -344.594,E2 -344.594} C_VEL
LIN {X 0,Y 608.48,Z 350.694,A -85,B 0,C 180,E1 -347.323,E2 -347.323} C_VEL
LIN {X 0,Y 608.451,Z 350.688,A -85,B 0,C 180,E1 -350.023,E2 -350.023} C_VEL
LIN {X 0,Y 608.481,Z 350.686,A -85,B 0,C 180,E1 -352.701,E2 -352.701} C_VEL
LIN {X 0,Y 608.462,Z 350.693,A -85,B 0,C 180,E1 -355.362,E2 -355.362} C_VEL
LIN {X 0,Y 608.448,Z 350.688,A -85,B 0,C 180,E1 -358.014,E2 -358.014} C_VEL
LIN {X 0,Y 608.482,Z 350.687,A -85,B 0,C 180,E1 -360.662,E2 -360.662} C_VEL
LIN {X 0,Y 608.486,Z 350.689,A -85,B 0,C 180,E1 -363.311,E2 -363.311} C_VEL
LIN {X 0,Y 608.452,Z 350.687,A -85,B 0,C 180,E1 -365.967,E2 -365.967} C_VEL
LIN {X 0,Y 608.46,Z 350.691,A -85,B 0,C 180,E1 -368.636,E2 -368.636} C_VEL
LIN {X 0,Y 608.477,Z 350.689,A -85,B 0,C 180,E1 -371.324,E2 -371.324} C_VEL
LIN {X 0,Y 608.458,Z 350.687,A -85,B 0,C 180,E1 -374.038,E2 -374.038} C_VEL
LIN {X 0,Y 608.477,Z 350.694,A -85,B 0,C 180,E1 -376.783,E2 -376.783} C_VEL
LIN {X 0,Y 608.451,Z 350.688,A -85,B 0,C 180,E1 -379.571,E2 -379.571} C_VEL
LIN {X 0,Y 608.485,Z 350.689,A -85,B 0,C 180,E1 -382.485,E2 -382.485} C_VEL
LIN {X 0,Y 608.45,Z 350.69,A -85,B 0,C 180,E1 -385.301,E2 -385.301} C_VEL
LIN {X 0,Y 608.445,Z 350.689,A -85,B 0,C 180,E1 -387.518,E2 -387.518} C_VEL
LIN {X 0,Y 608.46,Z 350.687,A -85,B 0,C 180,E1 -389.973,E2 -389.973} C_VEL
LIN {X 0,Y 608.467,Z 350.694,A -85,B 0,C 180,E1 -392.525,E2 -392.525} C_VEL
LIN {X 0,Y 608.441,Z 350.69,A -85,B 0,C 180,E1 -395.278,E2 -395.278} C_VEL
LIN {X 0,Y 608.468,Z 350.686,A -85,B 0,C 180,E1 -397.747,E2 -397.747} C_VEL
LIN {X 0,Y 608.476,Z 350.692,A -85,B 0,C 180,E1 -400.333,E2 -400.333} C_VEL
LIN {X 0,Y 608.483,Z 350.684,A -85,B 0,C 180,E1 -403.312,E2 -403.312} C_VEL
LIN {X 0,Y 608.468,Z 350.691,A -85,B 0,C 180,E1 -406.132,E2 -406.132} C_VEL
LIN {X 0,Y 608.456,Z 350.691,A -85,B 0,C 180,E1 -408.825,E2 -408.825} C_VEL
LIN {X 0,Y 608.469,Z 350.685,A -85,B 0,C 180,E1 -411.413,E2 -411.413} C_VEL
LIN {X 0,Y 608.477,Z 350.689,A -85,B 0,C 180,E1 -413.951,E2 -413.951} C_VEL
LIN {X 0,Y 608.464,Z 350.696,A -85,B 0,C 180,E1 -416.33,E2 -416.33} C_VEL
LIN {X 0,Y 608.477,Z 350.687,A -85,B 0,C 180,E1 -418.728,E2 -418.728} C_VEL
LIN {X 0,Y 608.469,Z 350.686,A -85,B 0,C 180,E1 -421.381,E2 -421.381} C_VEL
LIN {X 0,Y 608.474,Z 350.694,A -85,B 0,C 180,E1 -424.279,E2 -424.279} C_VEL
LIN {X 0,Y 608.45,Z 350.69,A -85,B 0,C 180,E1 -426.877,E2 -426.877} C_VEL
LIN {X 0,Y 608.503,Z 350.824,A -85,B 0,C 180,E1 -427.312,E2 -427.312} C_VEL
LIN {X 0,Y 608.567,Z 369.705,A -85,B 0,C 180,E1 -429.906,E2 -429.906} C_VEL
LIN {X 0,Y 608.521,Z 391.71,A -85,B 0,C 180,E1 -432.872,E2 -432.872} C_VEL
LIN {X 0,Y 608.476,Z 413.716,A -85,B 0,C 180,E1 -435.792,E2 -435.792} C_VEL
LIN {X 0,Y 608.504,Z 422.696,A -85,B 0,C 180,E1 -436.974,E2 -436.974} C_VEL
LIN {X 0,Y 608.538,Z 530.962,A -85,B 0,C 180,E1 -438.277,E2 -438.277} C_VEL
LIN {X 0,Y 608.514,Z 544.226,A -85,B 0,C 180,E1 -438.572,E2 -438.572} C_VEL
LIN {X 0,Y 608.517,Z 556.599,A -85,B 0,C 180,E1 -438.981,E2 -438.981} C_VEL
LIN {X 0,Y 608.498,Z 568.639,A -85,B 0,C 180,E1 -439.519,E2 -439.519} C_VEL
LIN {X 0,Y 608.48,Z 580.201,A -85,B 0,C 180,E1 -440.191,E2 -440.191} C_VEL
LIN {X 0,Y 608.485,Z 590.596,A -85,B 0,C 180,E1 -440.946,E2 -440.946} C_VEL
LIN {X 0,Y 608.475,Z 599.114,A -85,B 0,C 180,E1 -441.699,E2 -441.699} C_VEL
LIN {X 0,Y 608.471,Z 606.962,A -85,B 0,C 180,E1 -442.534,E2 -442.534} C_VEL
LIN {X 0,Y 608.461,Z 614.287,A -85,B 0,C 180,E1 -443.485,E2 -443.485} C_VEL
LIN {X 0,Y 608.45,Z 619.867,A -85,B 0,C 180,E1 -444.366,E2 -444.366} C_VEL
LIN {X 0,Y 608.432,Z 624.951,A -85,B 0,C 180,E1 -445.362,E2 -445.362} C_VEL
LIN {X 0,Y 608.449,Z 628.896,A -85,B 0,C 180,E1 -446.358,E2 -446.358} C_VEL
LIN {X 0,Y 608.425,Z 631.809,A -85,B 0,C 180,E1 -447.352,E2 -447.352} C_VEL
LIN {X 0,Y 608.442,Z 633.201,A -85,B 0,C 180,E1 -448.014,E2 -448.014} C_VEL
LIN {X 0,Y 608.438,Z 634.783,A -85,B 0,C 180,E1 -449.338,E2 -449.338} C_VEL
LIN {X 0,Y 608.434,Z 635,A -85,B 0,C 180,E1 -450,E2 -450} C_VEL
LIN {X 0,Y 608.448,Z 634.184,A -85,B 0,C 180,E1 -451.324,E2 -451.324} C_VEL
LIN {X 0,Y 608.442,Z 633.201,A -85,B 0,C 180,E1 -451.986,E2 -451.986} C_VEL
LIN {X 0,Y 608.425,Z 631.809,A -85,B 0,C 180,E1 -452.648,E2 -452.648} C_VEL
LIN {X 0,Y 608.449,Z 628.896,A -85,B 0,C 180,E1 -453.642,E2 -453.642} C_VEL
LIN {X 0,Y 608.432,Z 624.95,A -85,B 0,C 180,E1 -454.638,E2 -454.638} C_VEL
LIN {X 0,Y 608.437,Z 618.877,A -85,B 0,C 180,E1 -455.801,E2 -455.801} C_VEL
LIN {X 0,Y 608.462,Z 612.236,A -85,B 0,C 180,E1 -456.799,E2 -456.799} C_VEL
LIN {X 0,Y 608.455,Z 603.991,A -85,B 0,C 180,E1 -457.8,E2 -457.8} C_VEL
LIN {X 0,Y 608.472,Z 595.538,A -85,B 0,C 180,E1 -458.636,E2 -458.636} C_VEL
LIN {X 0,Y 608.471,Z 585.094,A -85,B 0,C 180,E1 -459.473,E2 -459.473} C_VEL
LIN {X 0,Y 608.494,Z 574.76,A -85,B 0,C 180,E1 -460.144,E2 -460.144} C_VEL
LIN {X 0,Y 608.521,Z 563.256,A -85,B 0,C 180,E1 -460.74,E2 -460.74} C_VEL
LIN {X 0,Y 608.531,Z 550.887,A -85,B 0,C 180,E1 -461.225,E2 -461.225} C_VEL
LIN {X 0,Y 608.537,Z 537.45,A -85,B 0,C 180,E1 -461.597,E2 -461.597} C_VEL
LIN {X 0,Y 608.546,Z 525.105,A -85,B 0,C 180,E1 -461.808,E2 -461.808} C_VEL
LIN {X 0,Y 608.493,Z 422.615,A -85,B 0,C 180,E1 -463.037,E2 -463.037} C_VEL
LIN {X 0,Y 608.497,Z 400.771,A -85,B 0,C 180,E1 -465.92,E2 -465.92} C_VEL
LIN {X 0,Y 608.517,Z 379.797,A -85,B 0,C 180,E1 -468.728,E2 -468.728} C_VEL
LIN {X 0,Y 608.557,Z 360.644,A -85,B 0,C 180,E1 -471.332,E2 -471.332} C_VEL
LIN {X 0,Y 608.457,Z 350.689,A -85,B 0,C 180,E1 -472.714,E2 -472.714} C_VEL
LIN {X 0,Y 608.45,Z 350.69,A -85,B 0,C 180,E1 -475.3,E2 -475.3} C_VEL
LIN {X 0,Y 608.449,Z 350.694,A -85,B 0,C 180,E1 -477.517,E2 -477.517} C_VEL
LIN {X 0,Y 608.472,Z 350.692,A -85,B 0,C 180,E1 -479.972,E2 -479.972} C_VEL
LIN {X 0,Y 608.455,Z 350.687,A -85,B 0,C 180,E1 -482.521,E2 -482.521} C_VEL
LIN {X 0,Y 608.454,Z 350.691,A -85,B 0,C 180,E1 -485.276,E2 -485.276} C_VEL
LIN {X 0,Y 608.467,Z 350.695,A -85,B 0,C 180,E1 -487.745,E2 -487.745} C_VEL
LIN {X 0,Y 608.445,Z 350.689,A -85,B 0,C 180,E1 -490.328,E2 -490.328} C_VEL
LIN {X 0,Y 608.473,Z 350.691,A -85,B 0,C 180,E1 -493.309,E2 -493.309} C_VEL
LIN {X 0,Y 608.468,Z 350.687,A -85,B 0,C 180,E1 -496.13,E2 -496.13} C_VEL
LIN {X 0,Y 608.455,Z 350.688,A -85,B 0,C 180,E1 -498.823,E2 -498.823} C_VEL
LIN {X 0,Y 608.468,Z 350.695,A -85,B 0,C 180,E1 -501.412,E2 -501.412} C_VEL
LIN {X 0,Y 608.471,Z 350.688,A -85,B 0,C 180,E1 -503.95,E2 -503.95} C_VEL
LIN {X 0,Y 608.461,Z 350.686,A -85,B 0,C 180,E1 -506.329,E2 -506.329} C_VEL
LIN {X 0,Y 608.473,Z 350.686,A -85,B 0,C 180,E1 -508.726,E2 -508.726} C_VEL
LIN {X 0,Y 608.478,Z 350.694,A -85,B 0,C 180,E1 -511.377,E2 -511.377} C_VEL
LIN {X 0,Y 608.446,Z 350.689,A -85,B 0,C 180,E1 -513.964,E2 -513.964} C_VEL
LIN {X 0,Y 608.46,Z 350.686,A -85,B 0,C 180,E1 -516.155,E2 -516.155} C_VEL
LIN {X 0,Y 608.47,Z 350.685,A -85,B 0,C 180,E1 -518.308,E2 -518.308} C_VEL
LIN {X 0,Y 608.472,Z 350.694,A -85,B 0,C 180,E1 -521.28,E2 -521.28} C_VEL
LIN {X 0,Y 608.457,Z 350.687,A -85,B 0,C 180,E1 -523.906,E2 -523.906} C_VEL
LIN {X 0,Y 608.466,Z 350.689,A -85,B 0,C 180,E1 -526.644,E2 -526.644} C_VEL
LIN {X 0,Y 608.473,Z 350.691,A -85,B 0,C 180,E1 -529.35,E2 -529.35} C_VEL
LIN {X 0,Y 608.47,Z 350.685,A -85,B 0,C 180,E1 -532.033,E2 -532.033} C_VEL
LIN {X 0,Y 608.471,Z 350.69,A -85,B 0,C 180,E1 -534.698,E2 -534.698} C_VEL
LIN {X 0,Y 608.484,Z 350.688,A -85,B 0,C 180,E1 -537.352,E2 -537.352} C_VEL
LIN {X 0,Y 608.468,Z 350.685,A -85,B 0,C 180,E1 -540,E2 -540} C_VEL
LIN {X 0,Y 608.486,Z 350.689,A -85,B 0,C 180,E1 -542.648,E2 -542.648} C_VEL
LIN {X 0,Y 608.469,Z 350.689,A -85,B 0,C 180,E1 -545.302,E2 -545.302} C_VEL
LIN {X 0,Y 608.471,Z 350.685,A -85,B 0,C 180,E1 -547.967,E2 -547.967} C_VEL
LIN {X 0,Y 608.456,Z 350.688,A -85,B 0,C 180,E1 -549.477,E2 -549.477} C_VEL
LIN {X 0,Y 607.774,Z 350.774,A -85,B 0,C 180,E1 -550.03,E2 -550.03} C_VEL
LIN {X 0,Y 604.916,Z 351.136,A -85,B 0,C 180,E1 -550.927,E2 -550.927} C_VEL
LIN {X 0,Y 602.515,Z 351.431,A -85,B 0,C 180,E1 -551.648,E2 -551.648} C_VEL
LIN {X 0,Y 601.489,Z 351.557,A -85,B 0,C 180,E1 -552.205,E2 -552.205} C_VEL
LIN {X 0,Y 601.408,Z 351.568,A -85,B 0,C 180,E1 -552.394,E2 -552.394} C_VEL
LIN {X 0,Y 601.432,Z 351.57,A -85,B 0,C 180,E1 -554.897,E2 -554.897} C_VEL
LIN {X 0,Y 601.432,Z 351.568,A -85,B 0,C 180,E1 -556.986,E2 -556.986} C_VEL
LIN {X 0,Y 601.404,Z 351.565,A -85,B 0,C 180,E1 -559.81,E2 -559.81} C_VEL
LIN {X 0,Y 601.448,Z 351.57,A -85,B 0,C 180,E1 -562.682,E2 -562.682} C_VEL
LIN {X 0,Y 601.401,Z 351.572,A -85,B 0,C 180,E1 -564.879,E2 -564.879} C_VEL
LIN {X 0,Y 601.419,Z 351.564,A -85,B 0,C 180,E1 -567.868,E2 -567.868} C_VEL
LIN {X 0,Y 601.42,Z 351.568,A -85,B 0,C 180,E1 -570.165,E2 -570.165} C_VEL
LIN {X 0,Y 601.426,Z 351.569,A -85,B 0,C 180,E1 -572.718,E2 -572.718} C_VEL
LIN {X 0,Y 601.391,Z 351.568,A -85,B 0,C 180,E1 -575.113,E2 -575.113} C_VEL
LIN {X 0,Y 601.43,Z 351.562,A -85,B 0,C 180,E1 -577.42,E2 -577.42} C_VEL
LIN {X 0,Y 601.406,Z 351.569,A -85,B 0,C 180,E1 -579.996,E2 -579.996} C_VEL
LIN {X 0,Y 601.434,Z 351.567,A -85,B 0,C 180,E1 -582.669,E2 -582.669} C_VEL
LIN {X 0,Y 601.422,Z 351.563,A -85,B 0,C 180,E1 -585.483,E2 -585.483} C_VEL
LIN {X 0,Y 601.42,Z 351.572,A -85,B 0,C 180,E1 -588.408,E2 -588.408} C_VEL
LIN {X 0,Y 601.434,Z 351.563,A -85,B 0,C 180,E1 -590.876,E2 -590.876} C_VEL
LIN {X 0,Y 601.441,Z 351.564,A -85,B 0,C 180,E1 -593.735,E2 -593.735} C_VEL
LIN {X 0,Y 601.431,Z 351.571,A -85,B 0,C 180,E1 -596.065,E2 -596.065} C_VEL
LIN {X 0,Y 601.429,Z 351.562,A -85,B 0,C 180,E1 -599.059,E2 -599.059} C_VEL
LIN {X 0,Y 601.429,Z 351.563,A -85,B 0,C 180,E1 -601.374,E2 -601.374} C_VEL
LIN {X 0,Y 601.401,Z 351.569,A -85,B 0,C 180,E1 -603.637,E2 -603.637} C_VEL
LIN {X 0,Y 601.453,Z 351.567,A -85,B 0,C 180,E1 -605.86,E2 -605.86} C_VEL
LIN {X 0,Y 601.405,Z 351.566,A -85,B 0,C 180,E1 -608.761,E2 -608.761} C_VEL
LIN {X 0,Y 601.462,Z 351.726,A -85,B 0,C 180,E1 -611.27,E2 -611.27} C_VEL
LIN {X 0,Y 601.487,Z 367.861,A -85,B 0,C 180,E1 -614.063,E2 -614.063} C_VEL
LIN {X 0,Y 601.413,Z 384.324,A -85,B 0,C 180,E1 -616.871,E2 -616.871} C_VEL
LIN {X 0,Y 601.68,Z 388.362,A -85,B 0,C 180,E1 -616.942,E2 -616.942} C_VEL
LIN {X 0,Y 601.615,Z 490.839,A -85,B 0,C 180,E1 -618.183,E2 -618.183} C_VEL
LIN {X 0,Y 601.562,Z 503.383,A -85,B 0,C 180,E1 -618.459,E2 -618.459} C_VEL
LIN {X 0,Y 601.541,Z 516.517,A -85,B 0,C 180,E1 -618.894,E2 -618.894} C_VEL
LIN {X 0,Y 601.517,Z 527.754,A -85,B 0,C 180,E1 -619.396,E2 -619.396} C_VEL
LIN {X 0,Y 601.485,Z 539.526,A -85,B 0,C 180,E1 -620.076,E2 -620.076} C_VEL
LIN {X 0,Y 601.444,Z 550.035,A -85,B 0,C 180,E1 -620.839,E2 -620.839} C_VEL
LIN {X 0,Y 601.429,Z 558.642,A -85,B 0,C 180,E1 -621.601,E2 -621.601} C_VEL
LIN {X 0,Y 601.418,Z 566.57,A -85,B 0,C 180,E1 -622.446,E2 -622.446} C_VEL
LIN {X 0,Y 601.376,Z 573.89,A -85,B 0,C 180,E1 -623.393,E2 -623.393} C_VEL
LIN {X 0,Y 601.372,Z 579.613,A -85,B 0,C 180,E1 -624.299,E2 -624.299} C_VEL
LIN {X 0,Y 601.336,Z 584.754,A -85,B 0,C 180,E1 -625.307,E2 -625.307} C_VEL
LIN {X 0,Y 601.367,Z 588.744,A -85,B 0,C 180,E1 -626.315,E2 -626.315} C_VEL
LIN {X 0,Y 601.324,Z 591.693,A -85,B 0,C 180,E1 -627.321,E2 -627.321} C_VEL
LIN {X 0,Y 601.343,Z 593.127,A -85,B 0,C 180,E1 -627.991,E2 -627.991} C_VEL
LIN {X 0,Y 601.339,Z 594.753,A -85,B 0,C 180,E1 -629.33,E2 -629.33} C_VEL
LIN {X 0,Y 601.336,Z 594.996,A -85,B 0,C 180,E1 -630,E2 -630} C_VEL
LIN {X 0,Y 601.339,Z 594.815,A -85,B 0,C 180,E1 -630.67,E2 -630.67} C_VEL
LIN {X 0,Y 601.343,Z 593.276,A -85,B 0,C 180,E1 -632.009,E2 -632.009} C_VEL
LIN {X 0,Y 601.326,Z 591.917,A -85,B 0,C 180,E1 -632.679,E2 -632.679} C_VEL
LIN {X 0,Y 601.368,Z 589.04,A -85,B 0,C 180,E1 -633.685,E2 -633.685} C_VEL
LIN {X 0,Y 601.337,Z 585.141,A -85,B 0,C 180,E1 -634.693,E2 -634.693} C_VEL
LIN {X 0,Y 601.373,Z 580.11,A -85,B 0,C 180,E1 -635.701,E2 -635.701} C_VEL
LIN {X 0,Y 601.382,Z 573.792,A -85,B 0,C 180,E1 -636.711,E2 -636.711} C_VEL
LIN {X 0,Y 601.396,Z 565.876,A -85,B 0,C 180,E1 -637.723,E2 -637.723} C_VEL
LIN {X 0,Y 601.436,Z 556.032,A -85,B 0,C 180,E1 -638.737,E2 -638.737} C_VEL
LIN {X 0,Y 601.45,Z 545.711,A -85,B 0,C 180,E1 -639.585,E2 -639.585} C_VEL
LIN {X 0,Y 601.487,Z 534.093,A -85,B 0,C 180,E1 -640.349,E2 -640.349} C_VEL
LIN {X 0,Y 601.549,Z 522.876,A -85,B 0,C 180,E1 -640.929,E2 -640.929} C_VEL
LIN {X 0,Y 601.55,Z 510.332,A -85,B 0,C 180,E1 -641.42,E2 -641.42} C_VEL
LIN {X 0,Y 601.587,Z 497.548,A -85,B 0,C 180,E1 -641.775,E2 -641.775} C_VEL
LIN {X 0,Y 601.601,Z 485.271,A -85,B 0,C 180,E1 -641.989,E2 -641.989} C_VEL
LIN {X 0,Y 601.52,Z 385.126,A -85,B 0,C 180,E1 -643.191,E2 -643.191} C_VEL
LIN {X 0,Y 601.421,Z 384.348,A -85,B 0,C 180,E1 -643.214,E2 -643.214} C_VEL
LIN {X 0,Y 601.472,Z 368.385,A -85,B 0,C 180,E1 -645.937,E2 -645.937} C_VEL
LIN {X 0,Y 601.509,Z 352.928,A -85,B 0,C 180,E1 -648.609,E2 -648.609} C_VEL
LIN {X 0,Y 601.427,Z 351.565,A -85,B 0,C 180,E1 -648.875,E2 -648.875} C_VEL
LIN {X 0,Y 601.408,Z 351.566,A -85,B 0,C 180,E1 -651.239,E2 -651.239} C_VEL
LIN {X 0,Y 601.462,Z 351.568,A -85,B 0,C 180,E1 -654.14,E2 -654.14} C_VEL
LIN {X 0,Y 601.448,Z 351.56,A -85,B 0,C 180,E1 -657.111,E2 -657.111} C_VEL
LIN {X 0,Y 601.423,Z 351.565,A -85,B 0,C 180,E1 -659.392,E2 -659.392} C_VEL
LIN {X 0,Y 601.412,Z 351.571,A -85,B 0,C 180,E1 -661.725,E2 -661.725} C_VEL
LIN {X 0,Y 601.429,Z 351.569,A -85,B 0,C 180,E1 -664.117,E2 -664.117} C_VEL
LIN {X 0,Y 601.411,Z 351.565,A -85,B 0,C 180,E1 -666.581,E2 -666.581} C_VEL
LIN {X 0,Y 601.44,Z 351.567,A -85,B 0,C 180,E1 -669.535,E2 -669.535} C_VEL
LIN {X 0,Y 601.406,Z 351.565,A -85,B 0,C 180,E1 -672.59,E2 -672.59} C_VEL
LIN {X 0,Y 601.421,Z 351.569,A -85,B 0,C 180,E1 -675.481,E2 -675.481} C_VEL
LIN {X 0,Y 601.422,Z 351.564,A -85,B 0,C 180,E1 -678.406,E2 -678.406} C_VEL
LIN {X 0,Y 601.43,Z 351.563,A -85,B 0,C 180,E1 -680.875,E2 -680.875} C_VEL
LIN {X 0,Y 601.437,Z 351.57,A -85,B 0,C 180,E1 -683.733,E2 -683.733} C_VEL
LIN {X 0,Y 601.426,Z 351.563,A -85,B 0,C 180,E1 -686.686,E2 -686.686} C_VEL
LIN {X 0,Y 601.426,Z 351.566,A -85,B 0,C 180,E1 -689.058,E2 -689.058} C_VEL
LIN {X 0,Y 601.434,Z 351.57,A -85,B 0,C 180,E1 -691.373,E2 -691.373} C_VEL
LIN {X 0,Y 601.402,Z 351.573,A -85,B 0,C 180,E1 -693.636,E2 -693.636} C_VEL
LIN {X 0,Y 601.417,Z 351.564,A -85,B 0,C 180,E1 -696.589,E2 -696.589} C_VEL
LIN {X 0,Y 601.431,Z 351.571,A -85,B 0,C 180,E1 -699.478,E2 -699.478} C_VEL
LIN {X 0,Y 601.397,Z 351.566,A -85,B 0,C 180,E1 -702.312,E2 -702.312} C_VEL
LIN {X 0,Y 601.414,Z 351.564,A -85,B 0,C 180,E1 -704.409,E2 -704.409} C_VEL
LIN {X 0,Y 601.424,Z 351.571,A -85,B 0,C 180,E1 -707.172,E2 -707.172} C_VEL
LIN {X 0,Y 601.43,Z 351.563,A -85,B 0,C 180,E1 -709.905,E2 -709.905} C_VEL
LIN {X 0,Y 601.448,Z 351.562,A -85,B 0,C 180,E1 -712.615,E2 -712.615} C_VEL
LIN {X 0,Y 601.429,Z 351.57,A -85,B 0,C 180,E1 -715.308,E2 -715.308} C_VEL
LIN {X 0,Y 601.419,Z 351.564,A -85,B 0,C 180,E1 -717.991,E2 -717.991} C_VEL
LIN {X 0,Y 601.452,Z 351.563,A -85,B 0,C 180,E1 -720.669,E2 -720.669} C_VEL
LIN {X 0,Y 601.437,Z 351.567,A -85,B 0,C 180,E1 -723.349,E2 -723.349} C_VEL
LIN {X 0,Y 601.405,Z 351.565,A -85,B 0,C 180,E1 -726.037,E2 -726.037} C_VEL
LIN {X 0,Y 601.439,Z 351.567,A -85,B 0,C 180,E1 -728.738,E2 -728.738} C_VEL
LIN {X 0,Y 601.431,Z 351.565,A -85,B 0,C 180,E1 -731.458,E2 -731.458} C_VEL
LIN {X 0,Y 601.411,Z 351.565,A -85,B 0,C 180,E1 -734.206,E2 -734.206} C_VEL
LIN {X 0,Y 601.431,Z 351.57,A -85,B 0,C 180,E1 -736.986,E2 -736.986} C_VEL
LIN {X 0,Y 601.405,Z 351.565,A -85,B 0,C 180,E1 -739.809,E2 -739.809} C_VEL
LIN {X 0,Y 601.448,Z 351.569,A -85,B 0,C 180,E1 -742.682,E2 -742.682} C_VEL
LIN {X 0,Y 601.402,Z 351.574,A -85,B 0,C 180,E1 -744.879,E2 -744.879} C_VEL
LIN {X 0,Y 601.42,Z 351.564,A -85,B 0,C 180,E1 -747.868,E2 -747.868} C_VEL
LIN {X 0,Y 601.42,Z 351.566,A -85,B 0,C 180,E1 -750.165,E2 -750.165} C_VEL
LIN {X 0,Y 601.427,Z 351.572,A -85,B 0,C 180,E1 -752.718,E2 -752.718} C_VEL
LIN {X 0,Y 601.41,Z 351.567,A -85,B 0,C 180,E1 -755.116,E2 -755.116} C_VEL
LIN {X 0,Y 601.431,Z 351.562,A -85,B 0,C 180,E1 -757.419,E2 -757.419} C_VEL
LIN {X 0,Y 601.409,Z 351.567,A -85,B 0,C 180,E1 -759.995,E2 -759.995} C_VEL
LIN {X 0,Y 601.435,Z 351.569,A -85,B 0,C 180,E1 -762.668,E2 -762.668} C_VEL
LIN {X 0,Y 601.421,Z 351.563,A -85,B 0,C 180,E1 -765.483,E2 -765.483} C_VEL
LIN {X 0,Y 601.423,Z 351.574,A -85,B 0,C 180,E1 -768.407,E2 -768.407} C_VEL
LIN {X 0,Y 601.436,Z 351.564,A -85,B 0,C 180,E1 -770.876,E2 -770.876} C_VEL
LIN {X 0,Y 601.442,Z 351.562,A -85,B 0,C 180,E1 -773.735,E2 -773.735} C_VEL
LIN {X 0,Y 601.433,Z 351.568,A -85,B 0,C 180,E1 -776.065,E2 -776.065} C_VEL
LIN {X 0,Y 601.43,Z 351.563,A -85,B 0,C 180,E1 -779.059,E2 -779.059} C_VEL
LIN {X 0,Y 601.429,Z 351.563,A -85,B 0,C 180,E1 -781.374,E2 -781.374} C_VEL
LIN {X 0,Y 601.402,Z 351.568,A -85,B 0,C 180,E1 -783.637,E2 -783.637} C_VEL
LIN {X 0,Y 601.419,Z 351.57,A -85,B 0,C 180,E1 -786.59,E2 -786.59} C_VEL
LIN {X 0,Y 601.419,Z 351.583,A -85,B 0,C 180,E1 -787.136,E2 -787.136} C_VEL
LIN {X 0,Y 601.673,Z 358.055,A -85,B 0,C 180,E1 -788.051,E2 -788.051} C_VEL
LIN {X 0,Y 601.602,Z 378.766,A -85,B 0,C 180,E1 -790.908,E2 -790.908} C_VEL
LIN {X 0,Y 601.52,Z 400.771,A -85,B 0,C 180,E1 -793.89,E2 -793.89} C_VEL
LIN {X 0,Y 601.475,Z 422.615,A -85,B 0,C 180,E1 -796.808,E2 -796.808} C_VEL
LIN {X 0,Y 601.691,Z 426.745,A -85,B 0,C 180,E1 -796.878,E2 -796.878} C_VEL
LIN {X 0,Y 601.605,Z 530.962,A -85,B 0,C 180,E1 -798.14,E2 -798.14} C_VEL
LIN {X 0,Y 601.574,Z 544.227,A -85,B 0,C 180,E1 -798.438,E2 -798.438} C_VEL
LIN {X 0,Y 601.54,Z 556.707,A -85,B 0,C 180,E1 -798.856,E2 -798.856} C_VEL
LIN {X 0,Y 601.523,Z 568.638,A -85,B 0,C 180,E1 -799.396,E2 -799.396} C_VEL
LIN {X 0,Y 601.481,Z 580.202,A -85,B 0,C 180,E1 -800.076,E2 -800.076} C_VEL
LIN {X 0,Y 601.444,Z 590.598,A -85,B 0,C 180,E1 -800.839,E2 -800.839} C_VEL
LIN {X 0,Y 601.429,Z 599.114,A -85,B 0,C 180,E1 -801.601,E2 -801.601} C_VEL
LIN {X 0,Y 601.418,Z 606.962,A -85,B 0,C 180,E1 -802.446,E2 -802.446} C_VEL
LIN {X 0,Y 601.37,Z 614.225,A -85,B 0,C 180,E1 -803.398,E2 -803.398} C_VEL
LIN {X 0,Y 601.372,Z 619.867,A -85,B 0,C 180,E1 -804.299,E2 -804.299} C_VEL
LIN {X 0,Y 601.337,Z 624.95,A -85,B 0,C 180,E1 -805.307,E2 -805.307} C_VEL
LIN {X 0,Y 601.367,Z 628.896,A -85,B 0,C 180,E1 -806.315,E2 -806.315} C_VEL
LIN {X 0,Y 601.325,Z 631.809,A -85,B 0,C 180,E1 -807.321,E2 -807.321} C_VEL
LIN {X 0,Y 601.341,Z 633.202,A -85,B 0,C 180,E1 -807.991,E2 -807.991} C_VEL
LIN {X 0,Y 601.339,Z 634.784,A -85,B 0,C 180,E1 -809.33,E2 -809.33} C_VEL
LIN {X 0,Y 601.335,Z 635,A -85,B 0,C 180,E1 -810,E2 -810} C_VEL
LIN {X 0,Y 601.348,Z 634.184,A -85,B 0,C 180,E1 -811.339,E2 -811.339} C_VEL
LIN {X 0,Y 601.341,Z 633.202,A -85,B 0,C 180,E1 -812.009,E2 -812.009} C_VEL
LIN {X 0,Y 601.325,Z 631.809,A -85,B 0,C 180,E1 -812.679,E2 -812.679} C_VEL
LIN {X 0,Y 601.367,Z 628.896,A -85,B 0,C 180,E1 -813.685,E2 -813.685} C_VEL
LIN {X 0,Y 601.337,Z 624.95,A -85,B 0,C 180,E1 -814.693,E2 -814.693} C_VEL
LIN {X 0,Y 601.372,Z 618.878,A -85,B 0,C 180,E1 -815.869,E2 -815.869} C_VEL
LIN {X 0,Y 601.382,Z 612.237,A -85,B 0,C 180,E1 -816.88,E2 -816.88} C_VEL
LIN {X 0,Y 601.4,Z 603.991,A -85,B 0,C 180,E1 -817.892,E2 -817.892} C_VEL
LIN {X 0,Y 601.436,Z 595.539,A -85,B 0,C 180,E1 -818.737,E2 -818.737} C_VEL
LIN {X 0,Y 601.442,Z 585.095,A -85,B 0,C 180,E1 -819.585,E2 -819.585} C_VEL
LIN {X 0,Y 601.472,Z 574.761,A -85,B 0,C 180,E1 -820.264,E2 -820.264} C_VEL
LIN {X 0,Y 601.536,Z 563.907,A -85,B 0,C 180,E1 -820.835,E2 -820.835} C_VEL
LIN {X 0,Y 601.556,Z 551.385,A -85,B 0,C 180,E1 -821.34,E2 -821.34} C_VEL
LIN {X 0,Y 601.568,Z 538.363,A -85,B 0,C 180,E1 -821.711,E2 -821.711} C_VEL
LIN {X 0,Y 601.614,Z 525.105,A -85,B 0,C 180,E1 -821.946,E2 -821.946} C_VEL
LIN {X 0,Y 601.517,Z 423.168,A -85,B 0,C 180,E1 -823.169,E2 -823.169} C_VEL
LIN {X 0,Y 601.472,Z 422.13,A -85,B 0,C 180,E1 -823.256,E2 -823.256} C_VEL
LIN {X 0,Y 601.526,Z 399.477,A -85,B 0,C 180,E1 -826.284,E2 -826.284} C_VEL
LIN {X 0,Y 601.603,Z 378.766,A -85,B 0,C 180,E1 -829.092,E2 -829.092} C_VEL
LIN {X 0,Y 601.671,Z 358.055,A -85,B 0,C 180,E1 -831.949,E2 -831.949} C_VEL
LIN {X 0,Y 601.419,Z 351.583,A -85,B 0,C 180,E1 -832.864,E2 -832.864} C_VEL
LIN {X 0,Y 601.401,Z 351.567,A -85,B 0,C 180,E1 -834.878,E2 -834.878} C_VEL
LIN {X 0,Y 601.418,Z 351.573,A -85,B 0,C 180,E1 -837.867,E2 -837.867} C_VEL
LIN {X 0,Y 601.428,Z 351.566,A -85,B 0,C 180,E1 -840.163,E2 -840.163} C_VEL
LIN {X 0,Y 601.417,Z 351.564,A -85,B 0,C 180,E1 -842.714,E2 -842.714} C_VEL
LIN {X 0,Y 601.421,Z 351.565,A -85,B 0,C 180,E1 -845.115,E2 -845.115} C_VEL
LIN {X 0,Y 601.433,Z 351.568,A -85,B 0,C 180,E1 -847.418,E2 -847.418} C_VEL
LIN {X 0,Y 601.409,Z 351.569,A -85,B 0,C 180,E1 -849.994,E2 -849.994} C_VEL
LIN {X 0,Y 601.407,Z 351.565,A -85,B 0,C 180,E1 -852.669,E2 -852.669} C_VEL
LIN {X 0,Y 601.421,Z 351.573,A -85,B 0,C 180,E1 -855.481,E2 -855.481} C_VEL
LIN {X 0,Y 601.423,Z 351.563,A -85,B 0,C 180,E1 -858.406,E2 -858.406} C_VEL
LIN {X 0,Y 601.433,Z 351.564,A -85,B 0,C 180,E1 -860.875,E2 -860.875} C_VEL
LIN {X 0,Y 601.439,Z 351.566,A -85,B 0,C 180,E1 -863.733,E2 -863.733} C_VEL
LIN {X 0,Y 601.426,Z 351.564,A -85,B 0,C 180,E1 -866.686,E2 -866.686} C_VEL
LIN {X 0,Y 601.428,Z 351.568,A -85,B 0,C 180,E1 -869.058,E2 -869.058} C_VEL
LIN {X 0,Y 601.437,Z 351.571,A -85,B 0,C 180,E1 -871.373,E2 -871.373} C_VEL
LIN {X 0,Y 601.404,Z 351.57,A -85,B 0,C 180,E1 -873.636,E2 -873.636} C_VEL
LIN {X 0,Y 601.419,Z 351.565,A -85,B 0,C 180,E1 -876.59,E2 -876.59} C_VEL
LIN {X 0,Y 601.434,Z 351.568,A -85,B 0,C 180,E1 -879.478,E2 -879.478} C_VEL
LIN {X 0,Y 601.398,Z 351.566,A -85,B 0,C 180,E1 -882.312,E2 -882.312} C_VEL
LIN {X 0,Y 601.414,Z 351.565,A -85,B 0,C 180,E1 -884.409,E2 -884.409} C_VEL
LIN {X 0,Y 601.425,Z 351.573,A -85,B 0,C 180,E1 -887.172,E2 -887.172} C_VEL
LIN {X 0,Y 601.43,Z 351.562,A -85,B 0,C 180,E1 -889.905,E2 -889.905} C_VEL
LIN {X 0,Y 601.45,Z 351.563,A -85,B 0,C 180,E1 -892.615,E2 -892.615} C_VEL
LIN {X 0,Y 601.428,Z 351.568,A -85,B 0,C 180,E1 -895.308,E2 -895.308} C_VEL
LIN {X 0,Y 601.418,Z 351.564,A -85,B 0,C 180,E1 -897.991,E2 -897.991} C_VEL
LIN {X 0,Y 601.456,Z 351.565,A -85,B 0,C 180,E1 -900.67,E2 -900.67} C_VEL
LIN {X 0,Y 601.433,Z 351.565,A -85,B 0,C 180,E1 -903.35,E2 -903.35} C_VEL
LIN {X 0,Y 601.405,Z 351.566,A -85,B 0,C 180,E1 -906.037,E2 -906.037} C_VEL
LIN {X 0,Y 601.438,Z 351.57,A -85,B 0,C 180,E1 -908.738,E2 -908.738} C_VEL
LIN {X 0,Y 601.43,Z 351.563,A -85,B 0,C 180,E1 -911.458,E2 -911.458} C_VEL
LIN {X 0,Y 601.408,Z 351.568,A -85,B 0,C 180,E1 -912.394,E2 -912.394} C_VEL
LIN {X 0,Y 600.749,Z 351.657,A -85,B 0,C 180,E1 -912.953,E2 -912.953} C_VEL
LIN {X 0,Y 597.899,Z 352.012,A -85,B 0,C 180,E1 -913.861,E2 -913.861} C_VEL
LIN {X 0,Y 595.486,Z 352.311,A -85,B 0,C 180,E1 -914.591,E2 -914.591} C_VEL
LIN {X 0,Y 594.447,Z 352.436,A -85,B 0,C 180,E1 -915.154,E2 -915.154} C_VEL
LIN {X 0,Y 594.361,Z 352.444,A -85,B 0,C 180,E1 -915.345,E2 -915.345} C_VEL
LIN {X 0,Y 594.377,Z 352.441,A -85,B 0,C 180,E1 -917.904,E2 -917.904} C_VEL
LIN {X 0,Y 594.381,Z 352.446,A -85,B 0,C 180,E1 -920.92,E2 -920.92} C_VEL
LIN {X 0,Y 594.386,Z 352.44,A -85,B 0,C 180,E1 -923.704,E2 -923.704} C_VEL
LIN {X 0,Y 594.384,Z 352.448,A -85,B 0,C 180,E1 -926.7,E2 -926.7} C_VEL
LIN {X 0,Y 594.38,Z 352.444,A -85,B 0,C 180,E1 -928.999,E2 -928.999} C_VEL
LIN {X 0,Y 594.388,Z 352.44,A -85,B 0,C 180,E1 -931.646,E2 -931.646} C_VEL
LIN {X 0,Y 594.375,Z 352.45,A -85,B 0,C 180,E1 -934.581,E2 -934.581} C_VEL
LIN {X 0,Y 594.381,Z 352.442,A -85,B 0,C 180,E1 -937.087,E2 -937.087} C_VEL
LIN {X 0,Y 594.369,Z 352.443,A -85,B 0,C 180,E1 -939.775,E2 -939.775} C_VEL
LIN {X 0,Y 594.384,Z 352.451,A -85,B 0,C 180,E1 -942.374,E2 -942.374} C_VEL
LIN {X 0,Y 594.359,Z 352.443,A -85,B 0,C 180,E1 -945.192,E2 -945.192} C_VEL
LIN {X 0,Y 594.378,Z 352.449,A -85,B 0,C 180,E1 -948.153,E2 -948.153} C_VEL
LIN {X 0,Y 594.385,Z 352.44,A -85,B 0,C 180,E1 -951.196,E2 -951.196} C_VEL
LIN {X 0,Y 594.394,Z 352.442,A -85,B 0,C 180,E1 -953.759,E2 -953.759} C_VEL
LIN {X 0,Y 594.376,Z 352.451,A -85,B 0,C 180,E1 -956.239,E2 -956.239} C_VEL
LIN {X 0,Y 594.39,Z 352.442,A -85,B 0,C 180,E1 -958.652,E2 -958.652} C_VEL
LIN {X 0,Y 594.383,Z 352.44,A -85,B 0,C 180,E1 -961.043,E2 -961.043} C_VEL
LIN {X 0,Y 594.386,Z 352.449,A -85,B 0,C 180,E1 -963.978,E2 -963.978} C_VEL
LIN {X 0,Y 594.377,Z 352.447,A -85,B 0,C 180,E1 -966.296,E2 -966.296} C_VEL
LIN {X 0,Y 594.403,Z 352.439,A -85,B 0,C 180,E1 -969.225,E2 -969.225} C_VEL
LIN {X 0,Y 594.413,Z 352.588,A -85,B 0,C 180,E1 -971.191,E2 -971.191} C_VEL
LIN {X 0,Y 594.459,Z 366.851,A -85,B 0,C 180,E1 -973.693,E2 -973.693} C_VEL
LIN {X 0,Y 594.394,Z 383.061,A -85,B 0,C 180,E1 -976.496,E2 -976.496} C_VEL
LIN {X 0,Y 594.387,Z 384.612,A -85,B 0,C 180,E1 -976.732,E2 -976.732} C_VEL
LIN {X 0,Y 594.763,Z 388.408,A -85,B 0,C 180,E1 -976.787,E2 -976.787} C_VEL
LIN {X 0,Y 594.669,Z 490.868,A -85,B 0,C 180,E1 -978.043,E2 -978.043} C_VEL
LIN {X 0,Y 594.617,Z 504.162,A -85,B 0,C 180,E1 -978.344,E2 -978.344} C_VEL
LIN {X 0,Y 594.56,Z 517.305,A -85,B 0,C 180,E1 -978.791,E2 -978.791} C_VEL
LIN {X 0,Y 594.519,Z 529.393,A -85,B 0,C 180,E1 -979.356,E2 -979.356} C_VEL
LIN {X 0,Y 594.474,Z 540.812,A -85,B 0,C 180,E1 -980.044,E2 -980.044} C_VEL
LIN {X 0,Y 594.406,Z 551.103,A -85,B 0,C 180,E1 -980.815,E2 -980.815} C_VEL
LIN {X 0,Y 594.373,Z 560.362,A -85,B 0,C 180,E1 -981.672,E2 -981.672} C_VEL
LIN {X 0,Y 594.317,Z 569.335,A -85,B 0,C 180,E1 -982.697,E2 -982.697} C_VEL
LIN {X 0,Y 594.285,Z 575.855,A -85,B 0,C 180,E1 -983.612,E2 -983.612} C_VEL
LIN {X 0,Y 594.289,Z 581.441,A -85,B 0,C 180,E1 -984.571,E2 -984.571} C_VEL
LIN {X 0,Y 594.27,Z 586.183,A -85,B 0,C 180,E1 -985.591,E2 -985.591} C_VEL
LIN {X 0,Y 594.267,Z 589.817,A -85,B 0,C 180,E1 -986.61,E2 -986.61} C_VEL
LIN {X 0,Y 594.225,Z 591.695,A -85,B 0,C 180,E1 -987.288,E2 -987.288} C_VEL
LIN {X 0,Y 594.242,Z 593.127,A -85,B 0,C 180,E1 -987.967,E2 -987.967} C_VEL
LIN {X 0,Y 594.24,Z 594.753,A -85,B 0,C 180,E1 -989.322,E2 -989.322} C_VEL
LIN {X 0,Y 594.236,Z 594.996,A -85,B 0,C 180,E1 -990,E2 -990} C_VEL
LIN {X 0,Y 594.239,Z 594.815,A -85,B 0,C 180,E1 -990.678,E2 -990.678} C_VEL
LIN {X 0,Y 594.242,Z 593.275,A -85,B 0,C 180,E1 -992.033,E2 -992.033} C_VEL
LIN {X 0,Y 594.226,Z 591.915,A -85,B 0,C 180,E1 -992.712,E2 -992.712} C_VEL
LIN {X 0,Y 594.289,Z 589.038,A -85,B 0,C 180,E1 -993.729,E2 -993.729} C_VEL
LIN {X 0,Y 594.242,Z 585.139,A -85,B 0,C 180,E1 -994.749,E2 -994.749} C_VEL
LIN {X 0,Y 594.299,Z 580.108,A -85,B 0,C 180,E1 -995.769,E2 -995.769} C_VEL
LIN {X 0,Y 594.316,Z 573.789,A -85,B 0,C 180,E1 -996.791,E2 -996.791} C_VEL
LIN {X 0,Y 594.346,Z 565.871,A -85,B 0,C 180,E1 -997.815,E2 -997.815} C_VEL
LIN {X 0,Y 594.381,Z 556.026,A -85,B 0,C 180,E1 -998.842,E2 -998.842} C_VEL
LIN {X 0,Y 594.433,Z 545.706,A -85,B 0,C 180,E1 -999.699,E2 -999.699} C_VEL
LIN {X 0,Y 594.505,Z 534.082,A -85,B 0,C 180,E1 -1000.472,E2 -1000.472} C_VEL
LIN {X 0,Y 594.564,Z 522.865,A -85,B 0,C 180,E1 -1001.059,E2 -1001.059} C_VEL
LIN {X 0,Y 594.587,Z 510.39,A -85,B 0,C 180,E1 -1001.553,E2 -1001.553} C_VEL
LIN {X 0,Y 594.643,Z 497.525,A -85,B 0,C 180,E1 -1001.915,E2 -1001.915} C_VEL
LIN {X 0,Y 594.681,Z 485.232,A -85,B 0,C 180,E1 -1002.13,E2 -1002.13} C_VEL
LIN {X 0,Y 594.666,Z 386.178,A -85,B 0,C 180,E1 -1003.332,E2 -1003.332} C_VEL
LIN {X 0,Y 594.383,Z 384.345,A -85,B 0,C 180,E1 -1003.374,E2 -1003.374} C_VEL
LIN {X 0,Y 594.441,Z 368.382,A -85,B 0,C 180,E1 -1006.131,E2 -1006.131} C_VEL
LIN {X 0,Y 594.509,Z 354.192,A -85,B 0,C 180,E1 -1008.613,E2 -1008.613} C_VEL
LIN {X 0,Y 594.396,Z 352.442,A -85,B 0,C 180,E1 -1008.932,E2 -1008.932} C_VEL
LIN {X 0,Y 594.368,Z 352.445,A -85,B 0,C 180,E1 -1011.503,E2 -1011.503} C_VEL
LIN {X 0,Y 594.391,Z 352.444,A -85,B 0,C 180,E1 -1014.445,E2 -1014.445} C_VEL
LIN {X 0,Y 594.383,Z 352.441,A -85,B 0,C 180,E1 -1016.699,E2 -1016.699} C_VEL
LIN {X 0,Y 594.382,Z 352.44,A -85,B 0,C 180,E1 -1018.998,E2 -1018.998} C_VEL
LIN {X 0,Y 594.391,Z 352.444,A -85,B 0,C 180,E1 -1021.644,E2 -1021.644} C_VEL
LIN {X 0,Y 594.398,Z 352.439,A -85,B 0,C 180,E1 -1024.578,E2 -1024.578} C_VEL
LIN {X 0,Y 594.383,Z 352.44,A -85,B 0,C 180,E1 -1027.086,E2 -1027.086} C_VEL
LIN {X 0,Y 594.374,Z 352.451,A -85,B 0,C 180,E1 -1029.774,E2 -1029.774} C_VEL
LIN {X 0,Y 594.363,Z 352.444,A -85,B 0,C 180,E1 -1032.375,E2 -1032.375} C_VEL
LIN {X 0,Y 594.359,Z 352.445,A -85,B 0,C 180,E1 -1035.19,E2 -1035.19} C_VEL
LIN {X 0,Y 594.368,Z 352.451,A -85,B 0,C 180,E1 -1037.624,E2 -1037.624} C_VEL
LIN {X 0,Y 594.386,Z 352.441,A -85,B 0,C 180,E1 -1040.32,E2 -1040.32} C_VEL
LIN {X 0,Y 594.381,Z 352.441,A -85,B 0,C 180,E1 -1042.913,E2 -1042.913} C_VEL
LIN {X 0,Y 594.378,Z 352.446,A -85,B 0,C 180,E1 -1045.86,E2 -1045.86} C_VEL
LIN {X 0,Y 594.385,Z 352.44,A -85,B 0,C 180,E1 -1048.65,E2 -1048.65} C_VEL
LIN {X 0,Y 594.381,Z 352.443,A -85,B 0,C 180,E1 -1051.04,E2 -1051.04} C_VEL
LIN {X 0,Y 594.383,Z 352.443,A -85,B 0,C 180,E1 -1053.975,E2 -1053.975} C_VEL
LIN {X 0,Y 594.385,Z 352.44,A -85,B 0,C 180,E1 -1056.296,E2 -1056.296} C_VEL
LIN {X 0,Y 594.403,Z 352.445,A -85,B 0,C 180,E1 -1059.224,E2 -1059.224} C_VEL
LIN {X 0,Y 594.377,Z 352.442,A -85,B 0,C 180,E1 -1062.096,E2 -1062.096} C_VEL
LIN {X 0,Y 594.367,Z 352.442,A -85,B 0,C 180,E1 -1064.219,E2 -1064.219} C_VEL
LIN {X 0,Y 594.37,Z 352.447,A -85,B 0,C 180,E1 -1067.017,E2 -1067.017} C_VEL
LIN {X 0,Y 594.391,Z 352.441,A -85,B 0,C 180,E1 -1069.784,E2 -1069.784} C_VEL
LIN {X 0,Y 594.412,Z 352.437,A -85,B 0,C 180,E1 -1072.527,E2 -1072.527} C_VEL
LIN {X 0,Y 594.397,Z 352.447,A -85,B 0,C 180,E1 -1075.252,E2 -1075.252} C_VEL
LIN {X 0,Y 594.389,Z 352.44,A -85,B 0,C 180,E1 -1077.967,E2 -1077.967} C_VEL
LIN {X 0,Y 594.422,Z 352.439,A -85,B 0,C 180,E1 -1080.677,E2 -1080.677} C_VEL
LIN {X 0,Y 594.387,Z 352.444,A -85,B 0,C 180,E1 -1083.389,E2 -1083.389} C_VEL
LIN {X 0,Y 594.361,Z 352.443,A -85,B 0,C 180,E1 -1086.109,E2 -1086.109} C_VEL
LIN {X 0,Y 594.411,Z 352.437,A -85,B 0,C 180,E1 -1088.157,E2 -1088.157} C_VEL
LIN {X 0,Y 594.39,Z 352.447,A -85,B 0,C 180,E1 -1091.08,E2 -1091.08} C_VEL
LIN {X 0,Y 594.378,Z 352.441,A -85,B 0,C 180,E1 -1093.679,E2 -1093.679} C_VEL
LIN {X 0,Y 594.394,Z 352.447,A -85,B 0,C 180,E1 -1096.723,E2 -1096.723} C_VEL
LIN {X 0,Y 594.365,Z 352.445,A -85,B 0,C 180,E1 -1099.335,E2 -1099.335} C_VEL
LIN {X 0,Y 594.366,Z 352.443,A -85,B 0,C 180,E1 -1101.503,E2 -1101.503} C_VEL
LIN {X 0,Y 594.386,Z 352.44,A -85,B 0,C 180,E1 -1103.704,E2 -1103.704} C_VEL
LIN {X 0,Y 594.385,Z 352.45,A -85,B 0,C 180,E1 -1106.7,E2 -1106.7} C_VEL
LIN {X 0,Y 594.382,Z 352.445,A -85,B 0,C 180,E1 -1108.999,E2 -1108.999} C_VEL
LIN {X 0,Y 594.388,Z 352.439,A -85,B 0,C 180,E1 -1111.646,E2 -1111.646} C_VEL
LIN {X 0,Y 594.392,Z 352.449,A -85,B 0,C 180,E1 -1114.579,E2 -1114.579} C_VEL
LIN {X 0,Y 594.383,Z 352.443,A -85,B 0,C 180,E1 -1117.087,E2 -1117.087} C_VEL
LIN {X 0,Y 594.372,Z 352.442,A -85,B 0,C 180,E1 -1119.775,E2 -1119.775} C_VEL
LIN {X 0,Y 594.385,Z 352.448,A -85,B 0,C 180,E1 -1122.374,E2 -1122.374} C_VEL
LIN {X 0,Y 594.359,Z 352.444,A -85,B 0,C 180,E1 -1125.192,E2 -1125.192} C_VEL
LIN {X 0,Y 594.364,Z 352.443,A -85,B 0,C 180,E1 -1127.625,E2 -1127.625} C_VEL
LIN {X 0,Y 594.392,Z 352.448,A -85,B 0,C 180,E1 -1130.322,E2 -1130.322} C_VEL
LIN {X 0,Y 594.384,Z 352.442,A -85,B 0,C 180,E1 -1132.914,E2 -1132.914} C_VEL
LIN {X 0,Y 594.384,Z 352.443,A -85,B 0,C 180,E1 -1135.861,E2 -1135.861} C_VEL
LIN {X 0,Y 594.39,Z 352.443,A -85,B 0,C 180,E1 -1138.652,E2 -1138.652} C_VEL
LIN {X 0,Y 594.383,Z 352.441,A -85,B 0,C 180,E1 -1141.043,E2 -1141.043} C_VEL
LIN {X 0,Y 594.388,Z 352.447,A -85,B 0,C 180,E1 -1143.977,E2 -1143.977} C_VEL
LIN {X 0,Y 594.386,Z 352.447,A -85,B 0,C 180,E1 -1146.666,E2 -1146.666} C_VEL
LIN {X 0,Y 594.403,Z 352.554,A -85,B 0,C 180,E1 -1146.989,E2 -1146.989} C_VEL
LIN {X 0,Y 594.768,Z 357.027,A -85,B 0,C 180,E1 -1147.638,E2 -1147.638} C_VEL
LIN {X 0,Y 594.674,Z 376.177,A -85,B 0,C 180,E1 -1150.317,E2 -1150.317} C_VEL
LIN {X 0,Y 594.534,Z 398.3,A -85,B 0,C 180,E1 -1153.358,E2 -1153.358} C_VEL
LIN {X 0,Y 594.447,Z 420.188,A -85,B 0,C 180,E1 -1156.323,E2 -1156.323} C_VEL
LIN {X 0,Y 594.451,Z 422.615,A -85,B 0,C 180,E1 -1156.65,E2 -1156.65} C_VEL
LIN {X 0,Y 594.785,Z 426.745,A -85,B 0,C 180,E1 -1156.722,E2 -1156.722} C_VEL
LIN {X 0,Y 594.656,Z 530.961,A -85,B 0,C 180,E1 -1157.999,E2 -1157.999} C_VEL
LIN {X 0,Y 594.617,Z 544.227,A -85,B 0,C 180,E1 -1158.301,E2 -1158.301} C_VEL
LIN {X 0,Y 594.589,Z 556.613,A -85,B 0,C 180,E1 -1158.72,E2 -1158.72} C_VEL
LIN {X 0,Y 594.537,Z 568.637,A -85,B 0,C 180,E1 -1159.27,E2 -1159.27} C_VEL
LIN {X 0,Y 594.469,Z 580.203,A -85,B 0,C 180,E1 -1159.958,E2 -1159.958} C_VEL
LIN {X 0,Y 594.413,Z 590.599,A -85,B 0,C 180,E1 -1160.73,E2 -1160.73} C_VEL
LIN {X 0,Y 594.383,Z 599.114,A -85,B 0,C 180,E1 -1161.501,E2 -1161.501} C_VEL
LIN {X 0,Y 594.347,Z 606.962,A -85,B 0,C 180,E1 -1162.356,E2 -1162.356} C_VEL
LIN {X 0,Y 594.282,Z 614.813,A -85,B 0,C 180,E1 -1163.408,E2 -1163.408} C_VEL
LIN {X 0,Y 594.289,Z 621.681,A -85,B 0,C 180,E1 -1164.571,E2 -1164.571} C_VEL
LIN {X 0,Y 594.27,Z 626.372,A -85,B 0,C 180,E1 -1165.591,E2 -1165.591} C_VEL
LIN {X 0,Y 594.267,Z 629.957,A -85,B 0,C 180,E1 -1166.61,E2 -1166.61} C_VEL
LIN {X 0,Y 594.226,Z 631.809,A -85,B 0,C 180,E1 -1167.288,E2 -1167.288} C_VEL
LIN {X 0,Y 594.24,Z 633.201,A -85,B 0,C 180,E1 -1167.967,E2 -1167.967} C_VEL
LIN {X 0,Y 594.239,Z 634.784,A -85,B 0,C 180,E1 -1169.322,E2 -1169.322} C_VEL
LIN {X 0,Y 594.236,Z 635,A -85,B 0,C 180,E1 -1170,E2 -1170} C_VEL
LIN {X 0,Y 594.247,Z 634.185,A -85,B 0,C 180,E1 -1171.355,E2 -1171.355} C_VEL
LIN {X 0,Y 594.24,Z 633.202,A -85,B 0,C 180,E1 -1172.033,E2 -1172.033} C_VEL
LIN {X 0,Y 594.226,Z 631.81,A -85,B 0,C 180,E1 -1172.712,E2 -1172.712} C_VEL
LIN {X 0,Y 594.288,Z 628.896,A -85,B 0,C 180,E1 -1173.729,E2 -1173.729} C_VEL
LIN {X 0,Y 594.242,Z 624.95,A -85,B 0,C 180,E1 -1174.749,E2 -1174.749} C_VEL
LIN {X 0,Y 594.304,Z 618.878,A -85,B 0,C 180,E1 -1175.939,E2 -1175.939} C_VEL
LIN {X 0,Y 594.308,Z 612.237,A -85,B 0,C 180,E1 -1176.962,E2 -1176.962} C_VEL
LIN {X 0,Y 594.359,Z 603.991,A -85,B 0,C 180,E1 -1177.986,E2 -1177.986} C_VEL
LIN {X 0,Y 594.382,Z 595.539,A -85,B 0,C 180,E1 -1178.842,E2 -1178.842} C_VEL
LIN {X 0,Y 594.427,Z 585.097,A -85,B 0,C 180,E1 -1179.699,E2 -1179.699} C_VEL
LIN {X 0,Y 594.482,Z 574.763,A -85,B 0,C 180,E1 -1180.386,E2 -1180.386} C_VEL
LIN {X 0,Y 594.559,Z 563.706,A -85,B 0,C 180,E1 -1180.974,E2 -1180.974} C_VEL
LIN {X 0,Y 594.582,Z 551.712,A -85,B 0,C 180,E1 -1181.464,E2 -1181.464} C_VEL
LIN {X 0,Y 594.637,Z 538.363,A -85,B 0,C 180,E1 -1181.85,E2 -1181.85} C_VEL
LIN {X 0,Y 594.693,Z 525.105,A -85,B 0,C 180,E1 -1182.087,E2 -1182.087} C_VEL
LIN {X 0,Y 594.642,Z 424.063,A -85,B 0,C 180,E1 -1183.313,E2 -1183.313} C_VEL
LIN {X 0,Y 594.431,Z 422.453,A -85,B 0,C 180,E1 -1183.373,E2 -1183.373} C_VEL
LIN {X 0,Y 594.523,Z 400.771,A -85,B 0,C 180,E1 -1186.305,E2 -1186.305} C_VEL
LIN {X 0,Y 594.636,Z 380.394,A -85,B 0,C 180,E1 -1189.099,E2 -1189.099} C_VEL
LIN {X 0,Y 594.801,Z 358.055,A -85,B 0,C 180,E1 -1192.216,E2 -1192.216} C_VEL
LIN {X 0,Y 594.664,Z 353.943,A -85,B 0,C 180,E1 -1192.803,E2 -1192.803} C_VEL
LIN {X 0,Y 594.392,Z 352.445,A -85,B 0,C 180,E1 -1193.058,E2 -1193.058} C_VEL
LIN {X 0,Y 594.376,Z 352.444,A -85,B 0,C 180,E1 -1195.192,E2 -1195.192} C_VEL
LIN {X 0,Y 594.386,Z 352.446,A -85,B 0,C 180,E1 -1197.526,E2 -1197.526} C_VEL
LIN {X 0,Y 594.388,Z 352.442,A -85,B 0,C 180,E1 -1200.328,E2 -1200.328} C_VEL
LIN {X 0,Y 594.377,Z 352.441,A -85,B 0,C 180,E1 -1202.949,E2 -1202.949} C_VEL
LIN {X 0,Y 594.385,Z 352.445,A -85,B 0,C 180,E1 -1205.406,E2 -1205.406} C_VEL
LIN {X 0,Y 594.384,Z 352.445,A -85,B 0,C 180,E1 -1207.94,E2 -1207.94} C_VEL
LIN {X 0,Y 594.376,Z 352.441,A -85,B 0,C 180,E1 -1210.822,E2 -1210.822} C_VEL
LIN {X 0,Y 594.378,Z 352.446,A -85,B 0,C 180,E1 -1213.84,E2 -1213.84} C_VEL
LIN {X 0,Y 594.382,Z 352.44,A -85,B 0,C 180,E1 -1216.702,E2 -1216.702} C_VEL
LIN {X 0,Y 594.385,Z 352.449,A -85,B 0,C 180,E1 -1219.434,E2 -1219.434} C_VEL
LIN {X 0,Y 594.386,Z 352.44,A -85,B 0,C 180,E1 -1222.39,E2 -1222.39} C_VEL
LIN {X 0,Y 594.379,Z 352.441,A -85,B 0,C 180,E1 -1224.671,E2 -1224.671} C_VEL
LIN {X 0,Y 594.375,Z 352.446,A -85,B 0,C 180,E1 -1227.087,E2 -1227.087} C_VEL
LIN {X 0,Y 594.394,Z 352.444,A -85,B 0,C 180,E1 -1229.668,E2 -1229.668} C_VEL
LIN {X 0,Y 594.383,Z 352.441,A -85,B 0,C 180,E1 -1232.539,E2 -1232.539} C_VEL
LIN {X 0,Y 594.373,Z 352.444,A -85,B 0,C 180,E1 -1234.807,E2 -1234.807} C_VEL
LIN {X 0,Y 594.397,Z 352.449,A -85,B 0,C 180,E1 -1237.254,E2 -1237.254} C_VEL
LIN {X 0,Y 594.375,Z 352.442,A -85,B 0,C 180,E1 -1239.946,E2 -1239.946} C_VEL
LIN {X 0,Y 594.388,Z 352.444,A -85,B 0,C 180,E1 -1242.807,E2 -1242.807} C_VEL
LIN {X 0,Y 594.379,Z 352.441,A -85,B 0,C 180,E1 -1245.825,E2 -1245.825} C_VEL
LIN {X 0,Y 594.388,Z 352.44,A -85,B 0,C 180,E1 -1248.404,E2 -1248.404} C_VEL
LIN {X 0,Y 594.398,Z 352.447,A -85,B 0,C 180,E1 -1251.158,E2 -1251.158} C_VEL
LIN {X 0,Y 594.398,Z 352.444,A -85,B 0,C 180,E1 -1253.299,E2 -1253.299} C_VEL
LIN {X 0,Y 594.355,Z 352.444,A -85,B 0,C 180,E1 -1255.932,E2 -1255.932} C_VEL
LIN {X 0,Y 594.389,Z 352.439,A -85,B 0,C 180,E1 -1257.967,E2 -1257.967} C_VEL
LIN {X 0,Y 594.425,Z 352.441,A -85,B 0,C 180,E1 -1260.677,E2 -1260.677} C_VEL
LIN {X 0,Y 594.384,Z 352.443,A -85,B 0,C 180,E1 -1263.389,E2 -1263.389} C_VEL
LIN {X 0,Y 594.361,Z 352.443,A -85,B 0,C 180,E1 -1266.109,E2 -1266.109} C_VEL
LIN {X 0,Y 594.411,Z 352.438,A -85,B 0,C 180,E1 -1268.157,E2 -1268.157} C_VEL
LIN {X 0,Y 594.391,Z 352.445,A -85,B 0,C 180,E1 -1271.081,E2 -1271.081} C_VEL
LIN {X 0,Y 594.378,Z 352.441,A -85,B 0,C 180,E1 -1273.679,E2 -1273.679} C_VEL
LIN {X 0,Y 594.361,Z 352.444,A -85,B 0,C 180,E1 -1275.345,E2 -1275.345} C_VEL
LIN {X 0,Y 593.691,Z 352.528,A -85,B 0,C 180,E1 -1275.911,E2 -1275.911} C_VEL
LIN {X 0,Y 590.835,Z 352.89,A -85,B 0,C 180,E1 -1276.829,E2 -1276.829} C_VEL
LIN {X 0,Y 588.429,Z 353.187,A -85,B 0,C 180,E1 -1277.568,E2 -1277.568} C_VEL
LIN {X 0,Y 587.402,Z 353.312,A -85,B 0,C 180,E1 -1278.138,E2 -1278.138} C_VEL
LIN {X 0,Y 587.322,Z 353.322,A -85,B 0,C 180,E1 -1278.331,E2 -1278.331} C_VEL
LIN {X 0,Y 587.349,Z 353.32,A -85,B 0,C 180,E1 -1281.045,E2 -1281.045} C_VEL
LIN {X 0,Y 587.359,Z 353.316,A -85,B 0,C 180,E1 -1283.257,E2 -1283.257} C_VEL
LIN {X 0,Y 587.356,Z 353.321,A -85,B 0,C 180,E1 -1286.278,E2 -1286.278} C_VEL
LIN {X 0,Y 587.347,Z 353.318,A -85,B 0,C 180,E1 -1289.135,E2 -1289.135} C_VEL
LIN {X 0,Y 587.352,Z 353.317,A -85,B 0,C 180,E1 -1291.839,E2 -1291.839} C_VEL
LIN {X 0,Y 587.343,Z 353.325,A -85,B 0,C 180,E1 -1294.349,E2 -1294.349} C_VEL
LIN {X 0,Y 587.347,Z 353.322,A -85,B 0,C 180,E1 -1296.747,E2 -1296.747} C_VEL
LIN {X 0,Y 587.34,Z 353.317,A -85,B 0,C 180,E1 -1299.36,E2 -1299.36} C_VEL
LIN {X 0,Y 587.332,Z 353.324,A -85,B 0,C 180,E1 -1302.109,E2 -1302.109} C_VEL
LIN {X 0,Y 587.312,Z 353.321,A -85,B 0,C 180,E1 -1305.09,E2 -1305.09} C_VEL
LIN {X 0,Y 587.32,Z 353.324,A -85,B 0,C 180,E1 -1307.926,E2 -1307.926} C_VEL
LIN {X 0,Y 587.344,Z 353.321,A -85,B 0,C 180,E1 -1310.642,E2 -1310.642} C_VEL
LIN {X 0,Y 587.352,Z 353.316,A -85,B 0,C 180,E1 -1313.292,E2 -1313.292} C_VEL
LIN {X 0,Y 587.367,Z 353.318,A -85,B 0,C 180,E1 -1315.781,E2 -1315.781} C_VEL
LIN {X 0,Y 587.351,Z 353.325,A -85,B 0,C 180,E1 -1318.232,E2 -1318.232} C_VEL
LIN {X 0,Y 587.35,Z 353.317,A -85,B 0,C 180,E1 -1320.867,E2 -1320.867} C_VEL
LIN {X 0,Y 587.36,Z 353.321,A -85,B 0,C 180,E1 -1323.82,E2 -1323.82} C_VEL
LIN {X 0,Y 587.33,Z 353.329,A -85,B 0,C 180,E1 -1325.994,E2 -1325.994} C_VEL
LIN {X 0,Y 587.32,Z 353.328,A -85,B 0,C 180,E1 -1328.226,E2 -1328.226} C_VEL
LIN {X 0,Y 587.376,Z 353.404,A -85,B 0,C 180,E1 -1331.102,E2 -1331.102} C_VEL
LIN {X 0,Y 587.446,Z 365.842,A -85,B 0,C 180,E1 -1333.314,E2 -1333.314} C_VEL
LIN {X 0,Y 587.369,Z 382.051,A -85,B 0,C 180,E1 -1336.155,E2 -1336.155} C_VEL
LIN {X 0,Y 587.358,Z 384.434,A -85,B 0,C 180,E1 -1336.568,E2 -1336.568} C_VEL
LIN {X 0,Y 587.851,Z 390.242,A -85,B 0,C 180,E1 -1336.651,E2 -1336.651} C_VEL
LIN {X 0,Y 587.731,Z 490.897,A -85,B 0,C 180,E1 -1337.899,E2 -1337.899} C_VEL
LIN {X 0,Y 587.685,Z 504.181,A -85,B 0,C 180,E1 -1338.205,E2 -1338.205} C_VEL
LIN {X 0,Y 587.595,Z 516.688,A -85,B 0,C 180,E1 -1338.632,E2 -1338.632} C_VEL
LIN {X 0,Y 587.553,Z 527.78,A -85,B 0,C 180,E1 -1339.141,E2 -1339.141} C_VEL
LIN {X 0,Y 587.48,Z 539.541,A -85,B 0,C 180,E1 -1339.837,E2 -1339.837} C_VEL
LIN {X 0,Y 587.393,Z 550.051,A -85,B 0,C 180,E1 -1340.618,E2 -1340.618} C_VEL
LIN {X 0,Y 587.323,Z 558.654,A -85,B 0,C 180,E1 -1341.398,E2 -1341.398} C_VEL
LIN {X 0,Y 587.274,Z 566.579,A -85,B 0,C 180,E1 -1342.263,E2 -1342.263} C_VEL
LIN {X 0,Y 587.235,Z 573.15,A -85,B 0,C 180,E1 -1343.127,E2 -1343.127} C_VEL
LIN {X 0,Y 587.237,Z 579.619,A -85,B 0,C 180,E1 -1344.161,E2 -1344.161} C_VEL
LIN {X 0,Y 587.147,Z 584.758,A -85,B 0,C 180,E1 -1345.194,E2 -1345.194} C_VEL
LIN {X 0,Y 587.213,Z 588.748,A -85,B 0,C 180,E1 -1346.226,E2 -1346.226} C_VEL
LIN {X 0,Y 587.131,Z 591.697,A -85,B 0,C 180,E1 -1347.256,E2 -1347.256} C_VEL
LIN {X 0,Y 587.14,Z 593.127,A -85,B 0,C 180,E1 -1347.942,E2 -1347.942} C_VEL
LIN {X 0,Y 587.14,Z 594.754,A -85,B 0,C 180,E1 -1349.314,E2 -1349.314} C_VEL
LIN {X 0,Y 587.137,Z 594.996,A -85,B 0,C 180,E1 -1350,E2 -1350} C_VEL
LIN {X 0,Y 587.14,Z 594.815,A -85,B 0,C 180,E1 -1350.686,E2 -1350.686} C_VEL
LIN {X 0,Y 587.141,Z 593.274,A -85,B 0,C 180,E1 -1352.058,E2 -1352.058} C_VEL
LIN {X 0,Y 587.133,Z 591.913,A -85,B 0,C 180,E1 -1352.744,E2 -1352.744} C_VEL
LIN {X 0,Y 587.213,Z 589.036,A -85,B 0,C 180,E1 -1353.774,E2 -1353.774} C_VEL
LIN {X 0,Y 587.147,Z 585.136,A -85,B 0,C 180,E1 -1354.806,E2 -1354.806} C_VEL
LIN {X 0,Y 587.229,Z 580.105,A -85,B 0,C 180,E1 -1355.839,E2 -1355.839} C_VEL
LIN {X 0,Y 587.23,Z 573.785,A -85,B 0,C 180,E1 -1356.873,E2 -1356.873} C_VEL
LIN {X 0,Y 587.288,Z 565.866,A -85,B 0,C 180,E1 -1357.91,E2 -1357.91} C_VEL
LIN {X 0,Y 587.343,Z 556.019,A -85,B 0,C 180,E1 -1358.949,E2 -1358.949} C_VEL
LIN {X 0,Y 587.42,Z 545.7,A -85,B 0,C 180,E1 -1359.816,E2 -1359.816} C_VEL
LIN {X 0,Y 587.49,Z 535.493,A -85,B 0,C 180,E1 -1360.511,E2 -1360.511} C_VEL
LIN {X 0,Y 587.576,Z 524.508,A -85,B 0,C 180,E1 -1361.111,E2 -1361.111} C_VEL
LIN {X 0,Y 587.624,Z 512.843,A -85,B 0,C 180,E1 -1361.607,E2 -1361.607} C_VEL
LIN {X 0,Y 587.677,Z 500.245,A -85,B 0,C 180,E1 -1361.992,E2 -1361.992} C_VEL
LIN {X 0,Y 587.743,Z 486.703,A -85,B 0,C 180,E1 -1362.254,E2 -1362.254} C_VEL
LIN {X 0,Y 587.729,Z 386.824,A -85,B 0,C 180,E1 -1363.484,E2 -1363.484} C_VEL
LIN {X 0,Y 587.363,Z 384.342,A -85,B 0,C 180,E1 -1363.537,E2 -1363.537} C_VEL
LIN {X 0,Y 587.443,Z 368.378,A -85,B 0,C 180,E1 -1366.328,E2 -1366.328} C_VEL
LIN {X 0,Y 587.469,Z 354.188,A -85,B 0,C 180,E1 -1368.844,E2 -1368.844} C_VEL
LIN {X 0,Y 587.361,Z 353.319,A -85,B 0,C 180,E1 -1369.044,E2 -1369.044} C_VEL
LIN {X 0,Y 587.324,Z 353.326,A -85,B 0,C 180,E1 -1371.774,E2 -1371.774} C_VEL
LIN {X 0,Y 587.353,Z 353.318,A -85,B 0,C 180,E1 -1374.758,E2 -1374.758} C_VEL
LIN {X 0,Y 587.352,Z 353.321,A -85,B 0,C 180,E1 -1377.692,E2 -1377.692} C_VEL
LIN {X 0,Y 587.342,Z 353.319,A -85,B 0,C 180,E1 -1380.51,E2 -1380.51} C_VEL
LIN {X 0,Y 587.338,Z 353.318,A -85,B 0,C 180,E1 -1383.111,E2 -1383.111} C_VEL
LIN {X 0,Y 587.355,Z 353.326,A -85,B 0,C 180,E1 -1385.895,E2 -1385.895} C_VEL
LIN {X 0,Y 587.33,Z 353.32,A -85,B 0,C 180,E1 -1388.478,E2 -1388.478} C_VEL
LIN {X 0,Y 587.333,Z 353.32,A -85,B 0,C 180,E1 -1391.156,E2 -1391.156} C_VEL
LIN {X 0,Y 587.322,Z 353.324,A -85,B 0,C 180,E1 -1394.113,E2 -1394.113} C_VEL
LIN {X 0,Y 587.319,Z 353.321,A -85,B 0,C 180,E1 -1396.994,E2 -1396.994} C_VEL
LIN {X 0,Y 587.314,Z 353.33,A -85,B 0,C 180,E1 -1399.745,E2 -1399.745} C_VEL
LIN {X 0,Y 587.341,Z 353.318,A -85,B 0,C 180,E1 -1402.392,E2 -1402.392} C_VEL
LIN {X 0,Y 587.342,Z 353.318,A -85,B 0,C 180,E1 -1404.945,E2 -1404.945} C_VEL
LIN {X 0,Y 587.338,Z 353.325,A -85,B 0,C 180,E1 -1407.421,E2 -1407.421} C_VEL
LIN {X 0,Y 587.328,Z 353.324,A -85,B 0,C 180,E1 -1409.829,E2 -1409.829} C_VEL
LIN {X 0,Y 587.344,Z 353.317,A -85,B 0,C 180,E1 -1412.306,E2 -1412.306} C_VEL
LIN {X 0,Y 587.33,Z 353.319,A -85,B 0,C 180,E1 -1414.483,E2 -1414.483} C_VEL
LIN {X 0,Y 587.362,Z 353.324,A -85,B 0,C 180,E1 -1417.487,E2 -1417.487} C_VEL
LIN {X 0,Y 587.339,Z 353.317,A -85,B 0,C 180,E1 -1420.425,E2 -1420.425} C_VEL
LIN {X 0,Y 587.351,Z 353.326,A -85,B 0,C 180,E1 -1423.311,E2 -1423.311} C_VEL
LIN {X 0,Y 587.353,Z 353.316,A -85,B 0,C 180,E1 -1426.154,E2 -1426.154} C_VEL
LIN {X 0,Y 587.343,Z 353.322,A -85,B 0,C 180,E1 -1428.962,E2 -1428.962} C_VEL
LIN {X 0,Y 587.365,Z 353.317,A -85,B 0,C 180,E1 -1431.745,E2 -1431.745} C_VEL
LIN {X 0,Y 587.356,Z 353.316,A -85,B 0,C 180,E1 -1434.507,E2 -1434.507} C_VEL
LIN {X 0,Y 587.379,Z 353.321,A -85,B 0,C 180,E1 -1437.257,E2 -1437.257} C_VEL
LIN {X 0,Y 587.373,Z 353.313,A -85,B 0,C 180,E1 -1440,E2 -1440} C_VEL
LIN {X 0,Y 587.377,Z 353.318,A -85,B 0,C 180,E1 -1442.743,E2 -1442.743} C_VEL
LIN {X 0,Y 587.358,Z 353.318,A -85,B 0,C 180,E1 -1445.493,E2 -1445.493} C_VEL
LIN {X 0,Y 587.365,Z 353.315,A -85,B 0,C 180,E1 -1448.255,E2 -1448.255} C_VEL
LIN {X 0,Y 587.352,Z 353.323,A -85,B 0,C 180,E1 -1451.142,E2 -1451.142} C_VEL
LIN {X 0,Y 587.355,Z 353.317,A -85,B 0,C 180,E1 -1454.261,E2 -1454.261} C_VEL
LIN {X 0,Y 587.354,Z 353.318,A -85,B 0,C 180,E1 -1457.406,E2 -1457.406} C_VEL
LIN {X 0,Y 587.331,Z 353.321,A -85,B 0,C 180,E1 -1460.305,E2 -1460.305} C_VEL
LIN {X 0,Y 587.36,Z 353.318,A -85,B 0,C 180,E1 -1463.257,E2 -1463.257} C_VEL
LIN {X 0,Y 587.356,Z 353.319,A -85,B 0,C 180,E1 -1466.278,E2 -1466.278} C_VEL
LIN {X 0,Y 587.348,Z 353.32,A -85,B 0,C 180,E1 -1469.135,E2 -1469.135} C_VEL
LIN {X 0,Y 587.352,Z 353.316,A -85,B 0,C 180,E1 -1471.839,E2 -1471.839} C_VEL
LIN {X 0,Y 587.352,Z 353.322,A -85,B 0,C 180,E1 -1474.35,E2 -1474.35} C_VEL
LIN {X 0,Y 587.348,Z 353.324,A -85,B 0,C 180,E1 -1476.747,E2 -1476.747} C_VEL
LIN {X 0,Y 587.341,Z 353.318,A -85,B 0,C 180,E1 -1479.36,E2 -1479.36} C_VEL
LIN {X 0,Y 587.332,Z 353.322,A -85,B 0,C 180,E1 -1482.109,E2 -1482.109} C_VEL
LIN {X 0,Y 587.311,Z 353.322,A -85,B 0,C 180,E1 -1485.09,E2 -1485.09} C_VEL
LIN {X 0,Y 587.349,Z 353.319,A -85,B 0,C 180,E1 -1487.928,E2 -1487.928} C_VEL
LIN {X 0,Y 587.333,Z 353.319,A -85,B 0,C 180,E1 -1491.059,E2 -1491.059} C_VEL
LIN {X 0,Y 587.352,Z 353.316,A -85,B 0,C 180,E1 -1493.292,E2 -1493.292} C_VEL
LIN {X 0,Y 587.367,Z 353.316,A -85,B 0,C 180,E1 -1495.781,E2 -1495.781} C_VEL
LIN {X 0,Y 587.351,Z 353.326,A -85,B 0,C 180,E1 -1498.233,E2 -1498.233} C_VEL
LIN {X 0,Y 587.35,Z 353.318,A -85,B 0,C 180,E1 -1500.867,E2 -1500.867} C_VEL
LIN {X 0,Y 587.361,Z 353.32,A -85,B 0,C 180,E1 -1503.819,E2 -1503.819} C_VEL
LIN {X 0,Y 587.338,Z 353.325,A -85,B 0,C 180,E1 -1506.743,E2 -1506.743} C_VEL
LIN {X 0,Y 587.379,Z 353.604,A -85,B 0,C 180,E1 -1506.849,E2 -1506.849} C_VEL
LIN {X 0,Y 587.857,Z 356.917,A -85,B 0,C 180,E1 -1507.345,E2 -1507.345} C_VEL
LIN {X 0,Y 587.743,Z 377.472,A -85,B 0,C 180,E1 -1510.257,E2 -1510.257} C_VEL
LIN {X 0,Y 587.553,Z 399.477,A -85,B 0,C 180,E1 -1513.317,E2 -1513.317} C_VEL
LIN {X 0,Y 587.43,Z 421.483,A -85,B 0,C 180,E1 -1516.333,E2 -1516.333} C_VEL
LIN {X 0,Y 587.396,Z 422.615,A -85,B 0,C 180,E1 -1516.486,E2 -1516.486} C_VEL
LIN {X 0,Y 587.89,Z 426.745,A -85,B 0,C 180,E1 -1516.564,E2 -1516.564} C_VEL
LIN {X 0,Y 587.712,Z 530.961,A -85,B 0,C 180,E1 -1517.855,E2 -1517.855} C_VEL
LIN {X 0,Y 587.668,Z 544.228,A -85,B 0,C 180,E1 -1518.161,E2 -1518.161} C_VEL
LIN {X 0,Y 587.621,Z 556.791,A -85,B 0,C 180,E1 -1518.591,E2 -1518.591} C_VEL
LIN {X 0,Y 587.552,Z 568.636,A -85,B 0,C 180,E1 -1519.141,E2 -1519.141} C_VEL
LIN {X 0,Y 587.465,Z 580.205,A -85,B 0,C 180,E1 -1519.837,E2 -1519.837} C_VEL
LIN {X 0,Y 587.391,Z 590.6,A -85,B 0,C 180,E1 -1520.618,E2 -1520.618} C_VEL
LIN {X 0,Y 587.321,Z 599.114,A -85,B 0,C 180,E1 -1521.398,E2 -1521.398} C_VEL
LIN {X 0,Y 587.273,Z 606.962,A -85,B 0,C 180,E1 -1522.263,E2 -1522.263} C_VEL
LIN {X 0,Y 587.23,Z 613.47,A -85,B 0,C 180,E1 -1523.126,E2 -1523.126} C_VEL
LIN {X 0,Y 587.236,Z 619.867,A -85,B 0,C 180,E1 -1524.161,E2 -1524.161} C_VEL
LIN {X 0,Y 587.147,Z 624.95,A -85,B 0,C 180,E1 -1525.194,E2 -1525.194} C_VEL
LIN {X 0,Y 587.212,Z 628.896,A -85,B 0,C 180,E1 -1526.226,E2 -1526.226} C_VEL
LIN {X 0,Y 587.132,Z 631.809,A -85,B 0,C 180,E1 -1527.256,E2 -1527.256} C_VEL
LIN {X 0,Y 587.139,Z 633.2,A -85,B 0,C 180,E1 -1527.942,E2 -1527.942} C_VEL
LIN {X 0,Y 587.14,Z 634.784,A -85,B 0,C 180,E1 -1529.314,E2 -1529.314} C_VEL
LIN {X 0,Y 587.137,Z 635,A -85,B 0,C 180,E1 -1530,E2 -1530} C_VEL
LIN {X 0,Y 587.147,Z 634.185,A -85,B 0,C 180,E1 -1531.372,E2 -1531.372} C_VEL
LIN {X 0,Y 587.139,Z 633.201,A -85,B 0,C 180,E1 -1532.058,E2 -1532.058} C_VEL
LIN {X 0,Y 587.132,Z 631.81,A -85,B 0,C 180,E1 -1532.744,E2 -1532.744} C_VEL
LIN {X 0,Y 587.212,Z 628.896,A -85,B 0,C 180,E1 -1533.774,E2 -1533.774} C_VEL
LIN {X 0,Y 587.147,Z 624.95,A -85,B 0,C 180,E1 -1534.806,E2 -1534.806} C_VEL
LIN {X 0,Y 587.217,Z 618.878,A -85,B 0,C 180,E1 -1536.011,E2 -1536.011} C_VEL
LIN {X 0,Y 587.245,Z 612.238,A -85,B 0,C 180,E1 -1537.046,E2 -1537.046} C_VEL
LIN {X 0,Y 587.299,Z 603.992,A -85,B 0,C 180,E1 -1538.083,E2 -1538.083} C_VEL
LIN {X 0,Y 587.343,Z 595.54,A -85,B 0,C 180,E1 -1538.949,E2 -1538.949} C_VEL
LIN {X 0,Y 587.416,Z 585.098,A -85,B 0,C 180,E1 -1539.816,E2 -1539.816} C_VEL
LIN {X 0,Y 587.496,Z 574.762,A -85,B 0,C 180,E1 -1540.511,E2 -1540.511} C_VEL
LIN {X 0,Y 587.583,Z 562.811,A -85,B 0,C 180,E1 -1541.149,E2 -1541.149} C_VEL
LIN {X 0,Y 587.624,Z 550.601,A -85,B 0,C 180,E1 -1541.639,E2 -1541.639} C_VEL
LIN {X 0,Y 587.696,Z 537.447,A -85,B 0,C 180,E1 -1542.014,E2 -1542.014} C_VEL
LIN {X 0,Y 587.774,Z 525.105,A -85,B 0,C 180,E1 -1542.231,E2 -1542.231} C_VEL
LIN {X 0,Y 587.725,Z 424.632,A -85,B 0,C 180,E1 -1543.466,E2 -1543.466} C_VEL
LIN {X 0,Y 587.396,Z 422.615,A -85,B 0,C 180,E1 -1543.514,E2 -1543.514} C_VEL
LIN {X 0,Y 587.547,Z 402.066,A -85,B 0,C 180,E1 -1546.325,E2 -1546.325} C_VEL
LIN {X 0,Y 587.686,Z 380.744,A -85,B 0,C 180,E1 -1549.285,E2 -1549.285} C_VEL
LIN {X 0,Y 587.903,Z 359.349,A -85,B 0,C 180,E1 -1552.305,E2 -1552.305} C_VEL
LIN {X 0,Y 587.644,Z 354.975,A -85,B 0,C 180,E1 -1552.943,E2 -1552.943} C_VEL
LIN {X 0,Y 587.336,Z 353.326,A -85,B 0,C 180,E1 -1553.205,E2 -1553.205} C_VEL
LIN {X 0,Y 587.336,Z 353.325,A -85,B 0,C 180,E1 -1555.516,E2 -1555.516} C_VEL
LIN {X 0,Y 587.348,Z 353.327,A -85,B 0,C 180,E1 -1557.817,E2 -1557.817} C_VEL
LIN {X 0,Y 587.342,Z 353.318,A -85,B 0,C 180,E1 -1560.51,E2 -1560.51} C_VEL
LIN {X 0,Y 587.338,Z 353.319,A -85,B 0,C 180,E1 -1563.111,E2 -1563.111} C_VEL
LIN {X 0,Y 587.356,Z 353.322,A -85,B 0,C 180,E1 -1565.895,E2 -1565.895} C_VEL
LIN {X 0,Y 587.331,Z 353.319,A -85,B 0,C 180,E1 -1568.478,E2 -1568.478} C_VEL
LIN {X 0,Y 587.334,Z 353.321,A -85,B 0,C 180,E1 -1571.156,E2 -1571.156} C_VEL
LIN {X 0,Y 587.33,Z 353.321,A -85,B 0,C 180,E1 -1574.113,E2 -1574.113} C_VEL
LIN {X 0,Y 587.333,Z 353.321,A -85,B 0,C 180,E1 -1576.995,E2 -1576.995} C_VEL
LIN {X 0,Y 587.322,Z 353.322,A -85,B 0,C 180,E1 -1579.98,E2 -1579.98} C_VEL
LIN {X 0,Y 587.341,Z 353.317,A -85,B 0,C 180,E1 -1582.392,E2 -1582.392} C_VEL
LIN {X 0,Y 587.345,Z 353.32,A -85,B 0,C 180,E1 -1584.945,E2 -1584.945} C_VEL
LIN {X 0,Y 587.338,Z 353.328,A -85,B 0,C 180,E1 -1587.421,E2 -1587.421} C_VEL
LIN {X 0,Y 587.34,Z 353.32,A -85,B 0,C 180,E1 -1589.83,E2 -1589.83} C_VEL
LIN {X 0,Y 587.344,Z 353.317,A -85,B 0,C 180,E1 -1592.306,E2 -1592.306} C_VEL
LIN {X 0,Y 587.331,Z 353.319,A -85,B 0,C 180,E1 -1594.483,E2 -1594.483} C_VEL
LIN {X 0,Y 587.362,Z 353.321,A -85,B 0,C 180,E1 -1597.487,E2 -1597.487} C_VEL
LIN {X 0,Y 587.34,Z 353.318,A -85,B 0,C 180,E1 -1600.425,E2 -1600.425} C_VEL
LIN {X 0,Y 587.35,Z 353.324,A -85,B 0,C 180,E1 -1603.311,E2 -1603.311} C_VEL
LIN {X 0,Y 587.353,Z 353.316,A -85,B 0,C 180,E1 -1606.154,E2 -1606.154} C_VEL
LIN {X 0,Y 587.342,Z 353.325,A -85,B 0,C 180,E1 -1608.962,E2 -1608.962} C_VEL
LIN {X 0,Y 587.364,Z 353.315,A -85,B 0,C 180,E1 -1611.745,E2 -1611.745} C_VEL
LIN {X 0,Y 587.358,Z 353.318,A -85,B 0,C 180,E1 -1614.507,E2 -1614.507} C_VEL
LIN {X 0,Y 587.378,Z 353.318,A -85,B 0,C 180,E1 -1617.257,E2 -1617.257} C_VEL
LIN {X 0,Y 587.373,Z 353.313,A -85,B 0,C 180,E1 -1620,E2 -1620} C_VEL
LIN {X 0,Y 587.378,Z 353.32,A -85,B 0,C 180,E1 -1622.743,E2 -1622.743} C_VEL
LIN {X 0,Y 587.357,Z 353.317,A -85,B 0,C 180,E1 -1625.493,E2 -1625.493} C_VEL
LIN {X 0,Y 587.365,Z 353.316,A -85,B 0,C 180,E1 -1628.255,E2 -1628.255} C_VEL
LIN {X 0,Y 587.352,Z 353.32,A -85,B 0,C 180,E1 -1631.142,E2 -1631.142} C_VEL
LIN {X 0,Y 587.355,Z 353.318,A -85,B 0,C 180,E1 -1634.261,E2 -1634.261} C_VEL
LIN {X 0,Y 587.354,Z 353.317,A -85,B 0,C 180,E1 -1637.406,E2 -1637.406} C_VEL
LIN {X 0,Y 587.322,Z 353.322,A -85,B 0,C 180,E1 -1638.331,E2 -1638.331} C_VEL
LIN {X 0,Y 586.668,Z 353.409,A -85,B 0,C 180,E1 -1638.903,E2 -1638.903} C_VEL
LIN {X 0,Y 583.832,Z 353.761,A -85,B 0,C 180,E1 -1639.831,E2 -1639.831} C_VEL
LIN {X 0,Y 581.422,Z 354.064,A -85,B 0,C 180,E1 -1640.578,E2 -1640.578} C_VEL
LIN {X 0,Y 580.374,Z 354.188,A -85,B 0,C 180,E1 -1641.155,E2 -1641.155} C_VEL
LIN {X 0,Y 580.282,Z 354.198,A -85,B 0,C 180,E1 -1641.35,E2 -1641.35} C_VEL
LIN {X 0,Y 580.295,Z 354.195,A -85,B 0,C 180,E1 -1643.557,E2 -1643.557} C_VEL
LIN {X 0,Y 580.321,Z 354.198,A -85,B 0,C 180,E1 -1646.342,E2 -1646.342} C_VEL
LIN {X 0,Y 580.298,Z 354.195,A -85,B 0,C 180,E1 -1649.311,E2 -1649.311} C_VEL
LIN {X 0,Y 580.299,Z 354.2,A -85,B 0,C 180,E1 -1652.201,E2 -1652.201} C_VEL
LIN {X 0,Y 580.284,Z 354.203,A -85,B 0,C 180,E1 -1654.697,E2 -1654.697} C_VEL
LIN {X 0,Y 580.295,Z 354.195,A -85,B 0,C 180,E1 -1657.269,E2 -1657.269} C_VEL
LIN {X 0,Y 580.293,Z 354.204,A -85,B 0,C 180,E1 -1660.272,E2 -1660.272} C_VEL
LIN {X 0,Y 580.287,Z 354.201,A -85,B 0,C 180,E1 -1662.706,E2 -1662.706} C_VEL
LIN {X 0,Y 580.266,Z 354.2,A -85,B 0,C 180,E1 -1665.61,E2 -1665.61} C_VEL
LIN {X 0,Y 580.277,Z 354.207,A -85,B 0,C 180,E1 -1668.232,E2 -1668.232} C_VEL
LIN {X 0,Y 580.287,Z 354.197,A -85,B 0,C 180,E1 -1670.967,E2 -1670.967} C_VEL
LIN {X 0,Y 580.295,Z 354.197,A -85,B 0,C 180,E1 -1673.599,E2 -1673.599} C_VEL
LIN {X 0,Y 580.318,Z 354.202,A -85,B 0,C 180,E1 -1676.146,E2 -1676.146} C_VEL
LIN {X 0,Y 580.287,Z 354.199,A -85,B 0,C 180,E1 -1678.616,E2 -1678.616} C_VEL
LIN {X 0,Y 580.293,Z 354.195,A -85,B 0,C 180,E1 -1681.025,E2 -1681.025} C_VEL
LIN {X 0,Y 580.292,Z 354.199,A -85,B 0,C 180,E1 -1683.667,E2 -1683.667} C_VEL
LIN {X 0,Y 580.299,Z 354.2,A -85,B 0,C 180,E1 -1685.684,E2 -1685.684} C_VEL
LIN {X 0,Y 580.271,Z 354.208,A -85,B 0,C 180,E1 -1687.948,E2 -1687.948} C_VEL
LIN {X 0,Y 580.329,Z 354.321,A -85,B 0,C 180,E1 -1691.03,E2 -1691.03} C_VEL
LIN {X 0,Y 580.463,Z 361.793,A -85,B 0,C 180,E1 -1692.381,E2 -1692.381} C_VEL
LIN {X 0,Y 580.384,Z 378.002,A -85,B 0,C 180,E1 -1695.269,E2 -1695.269} C_VEL
LIN {X 0,Y 580.329,Z 384.48,A -85,B 0,C 180,E1 -1696.402,E2 -1696.402} C_VEL
LIN {X 0,Y 580.961,Z 390.287,A -85,B 0,C 180,E1 -1696.49,E2 -1696.49} C_VEL
LIN {X 0,Y 580.79,Z 490.926,A -85,B 0,C 180,E1 -1697.752,E2 -1697.752} C_VEL
LIN {X 0,Y 580.74,Z 504.199,A -85,B 0,C 180,E1 -1698.062,E2 -1698.062} C_VEL
LIN {X 0,Y 580.651,Z 516.358,A -85,B 0,C 180,E1 -1698.481,E2 -1698.481} C_VEL
LIN {X 0,Y 580.558,Z 527.793,A -85,B 0,C 180,E1 -1699.009,E2 -1699.009} C_VEL
LIN {X 0,Y 580.481,Z 539.548,A -85,B 0,C 180,E1 -1699.713,E2 -1699.713} C_VEL
LIN {X 0,Y 580.345,Z 550.059,A -85,B 0,C 180,E1 -1700.503,E2 -1700.503} C_VEL
LIN {X 0,Y 580.272,Z 558.659,A -85,B 0,C 180,E1 -1701.292,E2 -1701.292} C_VEL
LIN {X 0,Y 580.222,Z 566.583,A -85,B 0,C 180,E1 -1702.168,E2 -1702.168} C_VEL
LIN {X 0,Y 580.168,Z 574.285,A -85,B 0,C 180,E1 -1703.21,E2 -1703.21} C_VEL
LIN {X 0,Y 580.139,Z 581.447,A -85,B 0,C 180,E1 -1704.439,E2 -1704.439} C_VEL
LIN {X 0,Y 580.108,Z 586.188,A -85,B 0,C 180,E1 -1705.484,E2 -1705.484} C_VEL
LIN {X 0,Y 580.123,Z 589.822,A -85,B 0,C 180,E1 -1706.527,E2 -1706.527} C_VEL
LIN {X 0,Y 580.043,Z 591.699,A -85,B 0,C 180,E1 -1707.222,E2 -1707.222} C_VEL
LIN {X 0,Y 580.04,Z 593.128,A -85,B 0,C 180,E1 -1707.917,E2 -1707.917} C_VEL
LIN {X 0,Y 580.041,Z 594.755,A -85,B 0,C 180,E1 -1709.306,E2 -1709.306} C_VEL
LIN {X 0,Y 580.038,Z 594.996,A -85,B 0,C 180,E1 -1710,E2 -1710} C_VEL
LIN {X 0,Y 580.04,Z 594.815,A -85,B 0,C 180,E1 -1710.694,E2 -1710.694} C_VEL
LIN {X 0,Y 580.04,Z 593.272,A -85,B 0,C 180,E1 -1712.083,E2 -1712.083} C_VEL
LIN {X 0,Y 580.044,Z 591.911,A -85,B 0,C 180,E1 -1712.778,E2 -1712.778} C_VEL
LIN {X 0,Y 580.11,Z 589.034,A -85,B 0,C 180,E1 -1713.82,E2 -1713.82} C_VEL
LIN {X 0,Y 580.054,Z 585.134,A -85,B 0,C 180,E1 -1714.865,E2 -1714.865} C_VEL
LIN {X 0,Y 580.162,Z 580.102,A -85,B 0,C 180,E1 -1715.91,E2 -1715.91} C_VEL
LIN {X 0,Y 580.158,Z 573.781,A -85,B 0,C 180,E1 -1716.958,E2 -1716.958} C_VEL
LIN {X 0,Y 580.241,Z 565.862,A -85,B 0,C 180,E1 -1718.007,E2 -1718.007} C_VEL
LIN {X 0,Y 580.308,Z 556.013,A -85,B 0,C 180,E1 -1719.058,E2 -1719.058} C_VEL
LIN {X 0,Y 580.42,Z 545.694,A -85,B 0,C 180,E1 -1719.936,E2 -1719.936} C_VEL
LIN {X 0,Y 580.495,Z 535.486,A -85,B 0,C 180,E1 -1720.639,E2 -1720.639} C_VEL
LIN {X 0,Y 580.644,Z 523.215,A -85,B 0,C 180,E1 -1721.31,E2 -1721.31} C_VEL
LIN {X 0,Y 580.67,Z 510.633,A -85,B 0,C 180,E1 -1721.825,E2 -1721.825} C_VEL
LIN {X 0,Y 580.742,Z 497.477,A -85,B 0,C 180,E1 -1722.204,E2 -1722.204} C_VEL
LIN {X 0,Y 580.814,Z 485.151,A -85,B 0,C 180,E1 -1722.424,E2 -1722.424} C_VEL
LIN {X 0,Y 580.84,Z 387.674,A -85,B 0,C 180,E1 -1723.636,E2 -1723.636} C_VEL
LIN {X 0,Y 580.307,Z 384.338,A -85,B 0,C 180,E1 -1723.704,E2 -1723.704} C_VEL
LIN {X 0,Y 580.448,Z 368.375,A -85,B 0,C 180,E1 -1726.531,E2 -1726.531} C_VEL
LIN {X 0,Y 580.463,Z 355.199,A -85,B 0,C 180,E1 -1728.897,E2 -1728.897} C_VEL
LIN {X 0,Y 580.322,Z 354.197,A -85,B 0,C 180,E1 -1729.085,E2 -1729.085} C_VEL
LIN {X 0,Y 580.276,Z 354.209,A -85,B 0,C 180,E1 -1732.052,E2 -1732.052} C_VEL
LIN {X 0,Y 580.308,Z 354.195,A -85,B 0,C 180,E1 -1735.079,E2 -1735.079} C_VEL
LIN {X 0,Y 580.301,Z 354.201,A -85,B 0,C 180,E1 -1738.185,E2 -1738.185} C_VEL
LIN {X 0,Y 580.292,Z 354.196,A -85,B 0,C 180,E1 -1740.695,E2 -1740.695} C_VEL
LIN {X 0,Y 580.303,Z 354.196,A -85,B 0,C 180,E1 -1743.316,E2 -1743.316} C_VEL
LIN {X 0,Y 580.325,Z 354.2,A -85,B 0,C 180,E1 -1745.767,E2 -1745.767} C_VEL
LIN {X 0,Y 580.287,Z 354.201,A -85,B 0,C 180,E1 -1748.145,E2 -1748.145} C_VEL
LIN {X 0,Y 580.296,Z 354.195,A -85,B 0,C 180,E1 -1750.842,E2 -1750.842} C_VEL
LIN {X 0,Y 580.275,Z 354.206,A -85,B 0,C 180,E1 -1753.657,E2 -1753.657} C_VEL
LIN {X 0,Y 580.282,Z 354.197,A -85,B 0,C 180,E1 -1756.607,E2 -1756.607} C_VEL
LIN {X 0,Y 580.296,Z 354.197,A -85,B 0,C 180,E1 -1759.156,E2 -1759.156} C_VEL
LIN {X 0,Y 580.286,Z 354.202,A -85,B 0,C 180,E1 -1761.926,E2 -1761.926} C_VEL
LIN {X 0,Y 580.299,Z 354.195,A -85,B 0,C 180,E1 -1764.456,E2 -1764.456} C_VEL
LIN {X 0,Y 580.288,Z 354.198,A -85,B 0,C 180,E1 -1766.975,E2 -1766.975} C_VEL
LIN {X 0,Y 580.296,Z 354.203,A -85,B 0,C 180,E1 -1769.425,E2 -1769.425} C_VEL
LIN {X 0,Y 580.313,Z 354.194,A -85,B 0,C 180,E1 -1772.136,E2 -1772.136} C_VEL
LIN {X 0,Y 580.3,Z 354.197,A -85,B 0,C 180,E1 -1774.92,E2 -1774.92} C_VEL
LIN {X 0,Y 580.321,Z 354.198,A -85,B 0,C 180,E1 -1777.199,E2 -1777.199} C_VEL
LIN {X 0,Y 580.301,Z 354.195,A -85,B 0,C 180,E1 -1780.177,E2 -1780.177} C_VEL
LIN {X 0,Y 580.321,Z 354.198,A -85,B 0,C 180,E1 -1783.103,E2 -1783.103} C_VEL
LIN {X 0,Y 580.318,Z 354.193,A -85,B 0,C 180,E1 -1785.983,E2 -1785.983} C_VEL
LIN {X 0,Y 580.322,Z 354.195,A -85,B 0,C 180,E1 -1788.827,E2 -1788.827} C_VEL
LIN {X 0,Y 580.328,Z 354.194,A -85,B 0,C 180,E1 -1791.644,E2 -1791.644} C_VEL
LIN {X 0,Y 580.321,Z 354.192,A -85,B 0,C 180,E1 -1794.44,E2 -1794.44} C_VEL
LIN {X 0,Y 580.343,Z 354.198,A -85,B 0,C 180,E1 -1797.223,E2 -1797.223} C_VEL
LIN {X 0,Y 580.343,Z 354.189,A -85,B 0,C 180,E1 -1800,E2 -1800} C_VEL
LIN {X 0,Y 580.342,Z 354.194,A -85,B 0,C 180,E1 -1802.776,E2 -1802.776} C_VEL
LIN {X 0,Y 580.322,Z 354.194,A -85,B 0,C 180,E1 -1805.56,E2 -1805.56} C_VEL
LIN {X 0,Y 580.329,Z 354.192,A -85,B 0,C 180,E1 -1808.356,E2 -1808.356} C_VEL
LIN {X 0,Y 580.323,Z 354.197,A -85,B 0,C 180,E1 -1811.209,E2 -1811.209} C_VEL
LIN {X 0,Y 580.318,Z 354.192,A -85,B 0,C 180,E1 -1814.017,E2 -1814.017} C_VEL
LIN {X 0,Y 580.309,Z 354.203,A -85,B 0,C 180,E1 -1816.916,E2 -1816.916} C_VEL
LIN {X 0,Y 580.302,Z 354.194,A -85,B 0,C 180,E1 -1819.822,E2 -1819.822} C_VEL
LIN {X 0,Y 580.322,Z 354.202,A -85,B 0,C 180,E1 -1822.801,E2 -1822.801} C_VEL
LIN {X 0,Y 580.301,Z 354.199,A -85,B 0,C 180,E1 -1825.08,E2 -1825.08} C_VEL
LIN {X 0,Y 580.313,Z 354.193,A -85,B 0,C 180,E1 -1827.864,E2 -1827.864} C_VEL
LIN {X 0,Y 580.287,Z 354.206,A -85,B 0,C 180,E1 -1830.697,E2 -1830.697} C_VEL
LIN {X 0,Y 580.299,Z 354.195,A -85,B 0,C 180,E1 -1833.318,E2 -1833.318} C_VEL
LIN {X 0,Y 580.32,Z 354.192,A -85,B 0,C 180,E1 -1835.768,E2 -1835.768} C_VEL
LIN {X 0,Y 580.284,Z 354.2,A -85,B 0,C 180,E1 -1838.147,E2 -1838.147} C_VEL
LIN {X 0,Y 580.301,Z 354.199,A -85,B 0,C 180,E1 -1840.843,E2 -1840.843} C_VEL
LIN {X 0,Y 580.287,Z 354.196,A -85,B 0,C 180,E1 -1843.657,E2 -1843.657} C_VEL
LIN {X 0,Y 580.281,Z 354.204,A -85,B 0,C 180,E1 -1846.609,E2 -1846.609} C_VEL
LIN {X 0,Y 580.297,Z 354.195,A -85,B 0,C 180,E1 -1849.158,E2 -1849.158} C_VEL
LIN {X 0,Y 580.288,Z 354.199,A -85,B 0,C 180,E1 -1851.928,E2 -1851.928} C_VEL
LIN {X 0,Y 580.308,Z 354.202,A -85,B 0,C 180,E1 -1854.458,E2 -1854.458} C_VEL
LIN {X 0,Y 580.29,Z 354.197,A -85,B 0,C 180,E1 -1856.976,E2 -1856.976} C_VEL
LIN {X 0,Y 580.302,Z 354.194,A -85,B 0,C 180,E1 -1859.426,E2 -1859.426} C_VEL
LIN {X 0,Y 580.299,Z 354.204,A -85,B 0,C 180,E1 -1862.142,E2 -1862.142} C_VEL
LIN {X 0,Y 580.322,Z 354.194,A -85,B 0,C 180,E1 -1865.27,E2 -1865.27} C_VEL
LIN {X 0,Y 580.331,Z 354.351,A -85,B 0,C 180,E1 -1866.66,E2 -1866.66} C_VEL
LIN {X 0,Y 580.968,Z 359.349,A -85,B 0,C 180,E1 -1867.414,E2 -1867.414} C_VEL
LIN {X 0,Y 580.785,Z 378.766,A -85,B 0,C 180,E1 -1870.195,E2 -1870.195} C_VEL
LIN {X 0,Y 580.569,Z 400.771,A -85,B 0,C 180,E1 -1873.292,E2 -1873.292} C_VEL
LIN {X 0,Y 580.392,Z 422.615,A -85,B 0,C 180,E1 -1876.32,E2 -1876.32} C_VEL
LIN {X 0,Y 580.981,Z 426.745,A -85,B 0,C 180,E1 -1876.401,E2 -1876.401} C_VEL
LIN {X 0,Y 580.785,Z 530.961,A -85,B 0,C 180,E1 -1877.708,E2 -1877.708} C_VEL
LIN {X 0,Y 580.726,Z 544.229,A -85,B 0,C 180,E1 -1878.017,E2 -1878.017} C_VEL
LIN {X 0,Y 580.65,Z 557.5,A -85,B 0,C 180,E1 -1878.481,E2 -1878.481} C_VEL
LIN {X 0,Y 580.554,Z 568.634,A -85,B 0,C 180,E1 -1879.009,E2 -1879.009} C_VEL
LIN {X 0,Y 580.444,Z 580.206,A -85,B 0,C 180,E1 -1879.712,E2 -1879.712} C_VEL
LIN {X 0,Y 580.341,Z 590.602,A -85,B 0,C 180,E1 -1880.503,E2 -1880.503} C_VEL
LIN {X 0,Y 580.271,Z 599.114,A -85,B 0,C 180,E1 -1881.292,E2 -1881.292} C_VEL
LIN {X 0,Y 580.221,Z 606.962,A -85,B 0,C 180,E1 -1882.168,E2 -1882.168} C_VEL
LIN {X 0,Y 580.153,Z 614.651,A -85,B 0,C 180,E1 -1883.222,E2 -1883.222} C_VEL
LIN {X 0,Y 580.139,Z 621.681,A -85,B 0,C 180,E1 -1884.439,E2 -1884.439} C_VEL
LIN {X 0,Y 580.108,Z 626.372,A -85,B 0,C 180,E1 -1885.484,E2 -1885.484} C_VEL
LIN {X 0,Y 580.123,Z 629.957,A -85,B 0,C 180,E1 -1886.527,E2 -1886.527} C_VEL
LIN {X 0,Y 580.043,Z 631.809,A -85,B 0,C 180,E1 -1887.222,E2 -1887.222} C_VEL
LIN {X 0,Y 580.038,Z 633.199,A -85,B 0,C 180,E1 -1887.917,E2 -1887.917} C_VEL
LIN {X 0,Y 580.04,Z 634.785,A -85,B 0,C 180,E1 -1889.306,E2 -1889.306} C_VEL
LIN {X 0,Y 580.037,Z 635,A -85,B 0,C 180,E1 -1890,E2 -1890} C_VEL
LIN {X 0,Y 580.047,Z 634.186,A -85,B 0,C 180,E1 -1891.389,E2 -1891.389} C_VEL
LIN {X 0,Y 580.038,Z 633.2,A -85,B 0,C 180,E1 -1892.083,E2 -1892.083} C_VEL
LIN {X 0,Y 580.043,Z 631.81,A -85,B 0,C 180,E1 -1892.778,E2 -1892.778} C_VEL
LIN {X 0,Y 580.109,Z 628.896,A -85,B 0,C 180,E1 -1893.82,E2 -1893.82} C_VEL
LIN {X 0,Y 580.054,Z 624.95,A -85,B 0,C 180,E1 -1894.865,E2 -1894.865} C_VEL
LIN {X 0,Y 580.139,Z 618.878,A -85,B 0,C 180,E1 -1896.085,E2 -1896.085} C_VEL
LIN {X 0,Y 580.184,Z 612.238,A -85,B 0,C 180,E1 -1897.132,E2 -1897.132} C_VEL
LIN {X 0,Y 580.25,Z 603.992,A -85,B 0,C 180,E1 -1898.182,E2 -1898.182} C_VEL
LIN {X 0,Y 580.308,Z 595.54,A -85,B 0,C 180,E1 -1899.058,E2 -1899.058} C_VEL
LIN {X 0,Y 580.417,Z 585.1,A -85,B 0,C 180,E1 -1899.936,E2 -1899.936} C_VEL
LIN {X 0,Y 580.507,Z 574.76,A -85,B 0,C 180,E1 -1900.639,E2 -1900.639} C_VEL
LIN {X 0,Y 580.597,Z 563.242,A -85,B 0,C 180,E1 -1901.264,E2 -1901.264} C_VEL
LIN {X 0,Y 580.664,Z 550.479,A -85,B 0,C 180,E1 -1901.785,E2 -1901.785} C_VEL
LIN {X 0,Y 580.768,Z 537.446,A -85,B 0,C 180,E1 -1902.159,E2 -1902.159} C_VEL
LIN {X 0,Y 580.845,Z 525.105,A -85,B 0,C 180,E1 -1902.379,E2 -1902.379} C_VEL
LIN {X 0,Y 580.8,Z 425.405,A -85,B 0,C 180,E1 -1903.62,E2 -1903.62} C_VEL
LIN {X 0,Y 580.392,Z 422.615,A -85,B 0,C 180,E1 -1903.68,E2 -1903.68} C_VEL
LIN {X 0,Y 580.568,Z 400.771,A -85,B 0,C 180,E1 -1906.708,E2 -1906.708} C_VEL
LIN {X 0,Y 580.785,Z 378.766,A -85,B 0,C 180,E1 -1909.805,E2 -1909.805} C_VEL
LIN {X 0,Y 580.968,Z 359.349,A -85,B 0,C 180,E1 -1912.586,E2 -1912.586} C_VEL
LIN {X 0,Y 580.312,Z 354.202,A -85,B 0,C 180,E1 -1913.377,E2 -1913.377} C_VEL
LIN {X 0,Y 580.294,Z 354.206,A -85,B 0,C 180,E1 -1915.848,E2 -1915.848} C_VEL
LIN {X 0,Y 580.301,Z 354.199,A -85,B 0,C 180,E1 -1918.185,E2 -1918.185} C_VEL
LIN {X 0,Y 580.292,Z 354.196,A -85,B 0,C 180,E1 -1920.695,E2 -1920.695} C_VEL
LIN {X 0,Y 580.303,Z 354.198,A -85,B 0,C 180,E1 -1923.316,E2 -1923.316} C_VEL
LIN {X 0,Y 580.326,Z 354.2,A -85,B 0,C 180,E1 -1925.767,E2 -1925.767} C_VEL
LIN {X 0,Y 580.287,Z 354.199,A -85,B 0,C 180,E1 -1928.145,E2 -1928.145} C_VEL
LIN {X 0,Y 580.297,Z 354.195,A -85,B 0,C 180,E1 -1930.842,E2 -1930.842} C_VEL
LIN {X 0,Y 580.283,Z 354.205,A -85,B 0,C 180,E1 -1933.656,E2 -1933.656} C_VEL
LIN {X 0,Y 580.288,Z 354.196,A -85,B 0,C 180,E1 -1936.607,E2 -1936.607} C_VEL
LIN {X 0,Y 580.301,Z 354.199,A -85,B 0,C 180,E1 -1939.157,E2 -1939.157} C_VEL
LIN {X 0,Y 580.286,Z 354.199,A -85,B 0,C 180,E1 -1941.926,E2 -1941.926} C_VEL
LIN {X 0,Y 580.301,Z 354.194,A -85,B 0,C 180,E1 -1944.456,E2 -1944.456} C_VEL
LIN {X 0,Y 580.287,Z 354.2,A -85,B 0,C 180,E1 -1946.975,E2 -1946.975} C_VEL
LIN {X 0,Y 580.303,Z 354.203,A -85,B 0,C 180,E1 -1949.425,E2 -1949.425} C_VEL
LIN {X 0,Y 580.313,Z 354.193,A -85,B 0,C 180,E1 -1952.136,E2 -1952.136} C_VEL
LIN {X 0,Y 580.301,Z 354.199,A -85,B 0,C 180,E1 -1954.92,E2 -1954.92} C_VEL
LIN {X 0,Y 580.322,Z 354.201,A -85,B 0,C 180,E1 -1957.199,E2 -1957.199} C_VEL
LIN {X 0,Y 580.302,Z 354.194,A -85,B 0,C 180,E1 -1960.178,E2 -1960.178} C_VEL
LIN {X 0,Y 580.321,Z 354.201,A -85,B 0,C 180,E1 -1963.103,E2 -1963.103} C_VEL
LIN {X 0,Y 580.318,Z 354.192,A -85,B 0,C 180,E1 -1965.983,E2 -1965.983} C_VEL
LIN {X 0,Y 580.322,Z 354.197,A -85,B 0,C 180,E1 -1968.827,E2 -1968.827} C_VEL
LIN {X 0,Y 580.328,Z 354.193,A -85,B 0,C 180,E1 -1971.644,E2 -1971.644} C_VEL
LIN {X 0,Y 580.322,Z 354.194,A -85,B 0,C 180,E1 -1974.44,E2 -1974.44} C_VEL
LIN {X 0,Y 580.343,Z 354.195,A -85,B 0,C 180,E1 -1977.224,E2 -1977.224} C_VEL
LIN {X 0,Y 580.343,Z 354.189,A -85,B 0,C 180,E1 -1980,E2 -1980} C_VEL
LIN {X 0,Y 580.343,Z 354.197,A -85,B 0,C 180,E1 -1982.777,E2 -1982.777} C_VEL
LIN {X 0,Y 580.321,Z 354.193,A -85,B 0,C 180,E1 -1985.56,E2 -1985.56} C_VEL
LIN {X 0,Y 580.328,Z 354.194,A -85,B 0,C 180,E1 -1988.356,E2 -1988.356} C_VEL
LIN {X 0,Y 580.323,Z 354.195,A -85,B 0,C 180,E1 -1991.209,E2 -1991.209} C_VEL
LIN {X 0,Y 580.318,Z 354.193,A -85,B 0,C 180,E1 -1994.017,E2 -1994.017} C_VEL
LIN {X 0,Y 580.309,Z 354.2,A -85,B 0,C 180,E1 -1996.917,E2 -1996.917} C_VEL
LIN {X 0,Y 580.302,Z 354.194,A -85,B 0,C 180,E1 -1999.823,E2 -1999.823} C_VEL
LIN {X 0,Y 580.282,Z 354.198,A -85,B 0,C 180,E1 -2001.35,E2 -2001.35} C_VEL
LIN {X 0,Y 579.593,Z 354.284,A -85,B 0,C 180,E1 -2001.929,E2 -2001.929} C_VEL
LIN {X 0,Y 576.72,Z 354.647,A -85,B 0,C 180,E1 -2002.87,E2 -2002.87} C_VEL
LIN {X 0,Y 574.321,Z 354.942,A -85,B 0,C 180,E1 -2003.626,E2 -2003.626} C_VEL
LIN {X 0,Y 573.316,Z 355.068,A -85,B 0,C 180,E1 -2004.21,E2 -2004.21} C_VEL
LIN {X 0,Y 573.247,Z 355.079,A -85,B 0,C 180,E1 -2004.408,E2 -2004.408} C_VEL
LIN {X 0,Y 573.258,Z 355.075,A -85,B 0,C 180,E1 -2006.976,E2 -2006.976} C_VEL
LIN {X 0,Y 573.243,Z 355.074,A -85,B 0,C 180,E1 -2009.49,E2 -2009.49} C_VEL
LIN {X 0,Y 573.252,Z 355.078,A -85,B 0,C 180,E1 -2012.23,E2 -2012.23} C_VEL
LIN {X 0,Y 573.234,Z 355.08,A -85,B 0,C 180,E1 -2014.773,E2 -2014.773} C_VEL
LIN {X 0,Y 573.249,Z 355.074,A -85,B 0,C 180,E1 -2017.167,E2 -2017.167} C_VEL
LIN {X 0,Y 573.242,Z 355.074,A -85,B 0,C 180,E1 -2019.608,E2 -2019.608} C_VEL
LIN {X 0,Y 573.246,Z 355.078,A -85,B 0,C 180,E1 -2022.644,E2 -2022.644} C_VEL
LIN {X 0,Y 573.231,Z 355.076,A -85,B 0,C 180,E1 -2025.667,E2 -2025.667} C_VEL
LIN {X 0,Y 573.227,Z 355.081,A -85,B 0,C 180,E1 -2028.544,E2 -2028.544} C_VEL
LIN {X 0,Y 573.247,Z 355.073,A -85,B 0,C 180,E1 -2031.3,E2 -2031.3} C_VEL
LIN {X 0,Y 573.264,Z 355.078,A -85,B 0,C 180,E1 -2034.012,E2 -2034.012} C_VEL
LIN {X 0,Y 573.268,Z 355.075,A -85,B 0,C 180,E1 -2036.519,E2 -2036.519} C_VEL
LIN {X 0,Y 573.238,Z 355.074,A -85,B 0,C 180,E1 -2039.117,E2 -2039.117} C_VEL
LIN {X 0,Y 573.253,Z 355.08,A -85,B 0,C 180,E1 -2041.971,E2 -2041.971} C_VEL
LIN {X 0,Y 573.255,Z 355.075,A -85,B 0,C 180,E1 -2044.591,E2 -2044.591} C_VEL
LIN {X 0,Y 573.235,Z 355.08,A -85,B 0,C 180,E1 -2047.663,E2 -2047.663} C_VEL
LIN {X 0,Y 573.268,Z 355.077,A -85,B 0,C 180,E1 -2050.671,E2 -2050.671} C_VEL
LIN {X 0,Y 573.283,Z 355.166,A -85,B 0,C 180,E1 -2050.942,E2 -2050.942} C_VEL
LIN {X 0,Y 573.444,Z 363.822,A -85,B 0,C 180,E1 -2052.527,E2 -2052.527} C_VEL
LIN {X 0,Y 573.342,Z 379.858,A -85,B 0,C 180,E1 -2055.415,E2 -2055.415} C_VEL
LIN {X 0,Y 573.283,Z 384.417,A -85,B 0,C 180,E1 -2056.229,E2 -2056.229} C_VEL
LIN {X 0,Y 574.081,Z 390.332,A -85,B 0,C 180,E1 -2056.325,E2 -2056.325} C_VEL
LIN {X 0,Y 573.877,Z 490.955,A -85,B 0,C 180,E1 -2057.603,E2 -2057.603} C_VEL
LIN {X 0,Y 573.8,Z 504.217,A -85,B 0,C 180,E1 -2057.915,E2 -2057.915} C_VEL
LIN {X 0,Y 573.712,Z 516.373,A -85,B 0,C 180,E1 -2058.339,E2 -2058.339} C_VEL
LIN {X 0,Y 573.594,Z 527.818,A -85,B 0,C 180,E1 -2058.874,E2 -2058.874} C_VEL
LIN {X 0,Y 573.447,Z 539.554,A -85,B 0,C 180,E1 -2059.586,E2 -2059.586} C_VEL
LIN {X 0,Y 573.332,Z 550.067,A -85,B 0,C 180,E1 -2060.386,E2 -2060.386} C_VEL
LIN {X 0,Y 573.241,Z 558.665,A -85,B 0,C 180,E1 -2061.185,E2 -2061.185} C_VEL
LIN {X 0,Y 573.161,Z 566.588,A -85,B 0,C 180,E1 -2062.071,E2 -2062.071} C_VEL
LIN {X 0,Y 573.093,Z 574.524,A -85,B 0,C 180,E1 -2063.163,E2 -2063.163} C_VEL
LIN {X 0,Y 573.071,Z 581.45,A -85,B 0,C 180,E1 -2064.37,E2 -2064.37} C_VEL
LIN {X 0,Y 573.029,Z 586.191,A -85,B 0,C 180,E1 -2065.428,E2 -2065.428} C_VEL
LIN {X 0,Y 573.022,Z 589.824,A -85,B 0,C 180,E1 -2066.484,E2 -2066.484} C_VEL
LIN {X 0,Y 572.959,Z 591.701,A -85,B 0,C 180,E1 -2067.188,E2 -2067.188} C_VEL
LIN {X 0,Y 572.939,Z 593.128,A -85,B 0,C 180,E1 -2067.891,E2 -2067.891} C_VEL
LIN {X 0,Y 572.941,Z 594.755,A -85,B 0,C 180,E1 -2069.297,E2 -2069.297} C_VEL
LIN {X 0,Y 572.939,Z 594.996,A -85,B 0,C 180,E1 -2070,E2 -2070} C_VEL
LIN {X 0,Y 572.94,Z 594.815,A -85,B 0,C 180,E1 -2070.703,E2 -2070.703} C_VEL
LIN {X 0,Y 572.94,Z 593.27,A -85,B 0,C 180,E1 -2072.109,E2 -2072.109} C_VEL
LIN {X 0,Y 572.96,Z 591.909,A -85,B 0,C 180,E1 -2072.812,E2 -2072.812} C_VEL
LIN {X 0,Y 573.015,Z 589.032,A -85,B 0,C 180,E1 -2073.868,E2 -2073.868} C_VEL
LIN {X 0,Y 572.963,Z 585.132,A -85,B 0,C 180,E1 -2074.926,E2 -2074.926} C_VEL
LIN {X 0,Y 573.075,Z 580.1,A -85,B 0,C 180,E1 -2075.983,E2 -2075.983} C_VEL
LIN {X 0,Y 573.083,Z 573.777,A -85,B 0,C 180,E1 -2077.044,E2 -2077.044} C_VEL
LIN {X 0,Y 573.175,Z 565.857,A -85,B 0,C 180,E1 -2078.106,E2 -2078.106} C_VEL
LIN {X 0,Y 573.287,Z 556.007,A -85,B 0,C 180,E1 -2079.17,E2 -2079.17} C_VEL
LIN {X 0,Y 573.423,Z 545.688,A -85,B 0,C 180,E1 -2080.058,E2 -2080.058} C_VEL
LIN {X 0,Y 573.555,Z 534.053,A -85,B 0,C 180,E1 -2080.859,E2 -2080.859} C_VEL
LIN {X 0,Y 573.657,Z 523.205,A -85,B 0,C 180,E1 -2081.449,E2 -2081.449} C_VEL
LIN {X 0,Y 573.727,Z 510.618,A -85,B 0,C 180,E1 -2081.97,E2 -2081.97} C_VEL
LIN {X 0,Y 573.8,Z 497.453,A -85,B 0,C 180,E1 -2082.354,E2 -2082.354} C_VEL
LIN {X 0,Y 573.898,Z 485.111,A -85,B 0,C 180,E1 -2082.577,E2 -2082.577} C_VEL
LIN {X 0,Y 573.929,Z 388.298,A -85,B 0,C 180,E1 -2083.795,E2 -2083.795} C_VEL
LIN {X 0,Y 573.266,Z 384.335,A -85,B 0,C 180,E1 -2083.876,E2 -2083.876} C_VEL
LIN {X 0,Y 573.417,Z 368.493,A -85,B 0,C 180,E1 -2086.717,E2 -2086.717} C_VEL
LIN {X 0,Y 573.475,Z 356.366,A -85,B 0,C 180,E1 -2088.922,E2 -2088.922} C_VEL
LIN {X 0,Y 573.278,Z 355.075,A -85,B 0,C 180,E1 -2089.18,E2 -2089.18} C_VEL
LIN {X 0,Y 573.232,Z 355.08,A -85,B 0,C 180,E1 -2091.58,E2 -2091.58} C_VEL
LIN {X 0,Y 573.277,Z 355.072,A -85,B 0,C 180,E1 -2094.633,E2 -2094.633} C_VEL
LIN {X 0,Y 573.251,Z 355.072,A -85,B 0,C 180,E1 -2096.975,E2 -2096.975} C_VEL
LIN {X 0,Y 573.248,Z 355.076,A -85,B 0,C 180,E1 -2099.488,E2 -2099.488} C_VEL
LIN {X 0,Y 573.254,Z 355.077,A -85,B 0,C 180,E1 -2102.228,E2 -2102.228} C_VEL
LIN {X 0,Y 573.251,Z 355.073,A -85,B 0,C 180,E1 -2104.773,E2 -2104.773} C_VEL
LIN {X 0,Y 573.252,Z 355.073,A -85,B 0,C 180,E1 -2107.165,E2 -2107.165} C_VEL
LIN {X 0,Y 573.246,Z 355.08,A -85,B 0,C 180,E1 -2109.606,E2 -2109.606} C_VEL
LIN {X 0,Y 573.236,Z 355.075,A -85,B 0,C 180,E1 -2112.641,E2 -2112.641} C_VEL
LIN {X 0,Y 573.235,Z 355.084,A -85,B 0,C 180,E1 -2115.666,E2 -2115.666} C_VEL
LIN {X 0,Y 573.24,Z 355.074,A -85,B 0,C 180,E1 -2118.544,E2 -2118.544} C_VEL
LIN {X 0,Y 573.243,Z 355.078,A -85,B 0,C 180,E1 -2121.298,E2 -2121.298} C_VEL
LIN {X 0,Y 573.258,Z 355.076,A -85,B 0,C 180,E1 -2124.01,E2 -2124.01} C_VEL
LIN {X 0,Y 573.278,Z 355.069,A -85,B 0,C 180,E1 -2126.518,E2 -2126.518} C_VEL
LIN {X 0,Y 573.232,Z 355.078,A -85,B 0,C 180,E1 -2129.115,E2 -2129.115} C_VEL
LIN {X 0,Y 573.258,Z 355.075,A -85,B 0,C 180,E1 -2131.968,E2 -2131.968} C_VEL
LIN {X 0,Y 573.248,Z 355.073,A -85,B 0,C 180,E1 -2134.589,E2 -2134.589} C_VEL
LIN {X 0,Y 573.251,Z 355.079,A -85,B 0,C 180,E1 -2137.663,E2 -2137.663} C_VEL
LIN {X 0,Y 573.271,Z 355.071,A -85,B 0,C 180,E1 -2140.727,E2 -2140.727} C_VEL
LIN {X 0,Y 573.253,Z 355.078,A -85,B 0,C 180,E1 -2143.622,E2 -2143.622} C_VEL
LIN {X 0,Y 573.232,Z 355.075,A -85,B 0,C 180,E1 -2146.529,E2 -2146.529} C_VEL
LIN {X 0,Y 573.269,Z 355.078,A -85,B 0,C 180,E1 -2149.403,E2 -2149.403} C_VEL
LIN {X 0,Y 573.282,Z 355.069,A -85,B 0,C 180,E1 -2152.25,E2 -2152.25} C_VEL
LIN {X 0,Y 573.308,Z 355.074,A -85,B 0,C 180,E1 -2155.077,E2 -2155.077} C_VEL
LIN {X 0,Y 573.301,Z 355.067,A -85,B 0,C 180,E1 -2157.892,E2 -2157.892} C_VEL
LIN {X 0,Y 573.331,Z 355.066,A -85,B 0,C 180,E1 -2160.702,E2 -2160.702} C_VEL
LIN {X 0,Y 573.24,Z 355.077,A -85,B 0,C 180,E1 -2163.514,E2 -2163.514} C_VEL
LIN {X 0,Y 573.288,Z 355.07,A -85,B 0,C 180,E1 -2165.628,E2 -2165.628} C_VEL
LIN {X 0,Y 573.3,Z 355.069,A -85,B 0,C 180,E1 -2168.459,E2 -2168.459} C_VEL
LIN {X 0,Y 573.289,Z 355.072,A -85,B 0,C 180,E1 -2171.312,E2 -2171.312} C_VEL
LIN {X 0,Y 573.272,Z 355.073,A -85,B 0,C 180,E1 -2174.425,E2 -2174.425} C_VEL
LIN {X 0,Y 573.253,Z 355.078,A -85,B 0,C 180,E1 -2177.112,E2 -2177.112} C_VEL
LIN {X 0,Y 573.253,Z 355.073,A -85,B 0,C 180,E1 -2180.077,E2 -2180.077} C_VEL
LIN {X 0,Y 573.263,Z 355.075,A -85,B 0,C 180,E1 -2183.154,E2 -2183.154} C_VEL
LIN {X 0,Y 573.282,Z 355.071,A -85,B 0,C 180,E1 -2186.189,E2 -2186.189} C_VEL
LIN {X 0,Y 573.238,Z 355.082,A -85,B 0,C 180,E1 -2188.565,E2 -2188.565} C_VEL
LIN {X 0,Y 573.231,Z 355.08,A -85,B 0,C 180,E1 -2190.993,E2 -2190.993} C_VEL
LIN {X 0,Y 573.282,Z 355.069,A -85,B 0,C 180,E1 -2193.529,E2 -2193.529} C_VEL
LIN {X 0,Y 573.255,Z 355.074,A -85,B 0,C 180,E1 -2196.049,E2 -2196.049} C_VEL
LIN {X 0,Y 573.244,Z 355.081,A -85,B 0,C 180,E1 -2198.702,E2 -2198.702} C_VEL
LIN {X 0,Y 573.25,Z 355.073,A -85,B 0,C 180,E1 -2201.597,E2 -2201.597} C_VEL
LIN {X 0,Y 573.235,Z 355.082,A -85,B 0,C 180,E1 -2204.334,E2 -2204.334} C_VEL
LIN {X 0,Y 573.239,Z 355.074,A -85,B 0,C 180,E1 -2207.359,E2 -2207.359} C_VEL
LIN {X 0,Y 573.246,Z 355.084,A -85,B 0,C 180,E1 -2210.394,E2 -2210.394} C_VEL
LIN {X 0,Y 573.254,Z 355.073,A -85,B 0,C 180,E1 -2213.079,E2 -2213.079} C_VEL
LIN {X 0,Y 573.273,Z 355.071,A -85,B 0,C 180,E1 -2215.673,E2 -2215.673} C_VEL
LIN {X 0,Y 573.248,Z 355.082,A -85,B 0,C 180,E1 -2218.186,E2 -2218.186} C_VEL
LIN {X 0,Y 573.265,Z 355.076,A -85,B 0,C 180,E1 -2220.635,E2 -2220.635} C_VEL
LIN {X 0,Y 573.251,Z 355.075,A -85,B 0,C 180,E1 -2223.025,E2 -2223.025} C_VEL
LIN {X 0,Y 573.276,Z 355.073,A -85,B 0,C 180,E1 -2225.367,E2 -2225.367} C_VEL
LIN {X 0,Y 573.275,Z 355.243,A -85,B 0,C 180,E1 -2226.503,E2 -2226.503} C_VEL
LIN {X 0,Y 574.055,Z 360.64,A -85,B 0,C 180,E1 -2227.317,E2 -2227.317} C_VEL
LIN {X 0,Y 573.838,Z 380.062,A -85,B 0,C 180,E1 -2230.132,E2 -2230.132} C_VEL
LIN {X 0,Y 573.572,Z 402.12,A -85,B 0,C 180,E1 -2233.273,E2 -2233.273} C_VEL
LIN {X 0,Y 573.4,Z 422.615,A -85,B 0,C 180,E1 -2236.15,E2 -2236.15} C_VEL
LIN {X 0,Y 574.102,Z 428.534,A -85,B 0,C 180,E1 -2236.257,E2 -2236.257} C_VEL
LIN {X 0,Y 573.875,Z 530.961,A -85,B 0,C 180,E1 -2237.558,E2 -2237.558} C_VEL
LIN {X 0,Y 573.78,Z 544.229,A -85,B 0,C 180,E1 -2237.87,E2 -2237.87} C_VEL
LIN {X 0,Y 573.709,Z 556.381,A -85,B 0,C 180,E1 -2238.294,E2 -2238.294} C_VEL
LIN {X 0,Y 573.574,Z 567.588,A -85,B 0,C 180,E1 -2238.817,E2 -2238.817} C_VEL
LIN {X 0,Y 573.469,Z 578.914,A -85,B 0,C 180,E1 -2239.497,E2 -2239.497} C_VEL
LIN {X 0,Y 573.345,Z 589.544,A -85,B 0,C 180,E1 -2240.297,E2 -2240.297} C_VEL
LIN {X 0,Y 573.241,Z 599.115,A -85,B 0,C 180,E1 -2241.185,E2 -2241.185} C_VEL
LIN {X 0,Y 573.161,Z 606.962,A -85,B 0,C 180,E1 -2242.071,E2 -2242.071} C_VEL
LIN {X 0,Y 573.072,Z 614.955,A -85,B 0,C 180,E1 -2243.186,E2 -2243.186} C_VEL
LIN {X 0,Y 573.07,Z 621.681,A -85,B 0,C 180,E1 -2244.37,E2 -2244.37} C_VEL
LIN {X 0,Y 573.029,Z 626.372,A -85,B 0,C 180,E1 -2245.428,E2 -2245.428} C_VEL
LIN {X 0,Y 573.022,Z 629.957,A -85,B 0,C 180,E1 -2246.484,E2 -2246.484} C_VEL
LIN {X 0,Y 572.959,Z 631.808,A -85,B 0,C 180,E1 -2247.188,E2 -2247.188} C_VEL
LIN {X 0,Y 572.938,Z 633.198,A -85,B 0,C 180,E1 -2247.891,E2 -2247.891} C_VEL
LIN {X 0,Y 572.941,Z 634.785,A -85,B 0,C 180,E1 -2249.297,E2 -2249.297} C_VEL
LIN {X 0,Y 572.938,Z 635,A -85,B 0,C 180,E1 -2250,E2 -2250} C_VEL
LIN {X 0,Y 572.946,Z 634.186,A -85,B 0,C 180,E1 -2251.406,E2 -2251.406} C_VEL
LIN {X 0,Y 572.938,Z 633.2,A -85,B 0,C 180,E1 -2252.109,E2 -2252.109} C_VEL
LIN {X 0,Y 572.959,Z 631.81,A -85,B 0,C 180,E1 -2252.812,E2 -2252.812} C_VEL
LIN {X 0,Y 573.014,Z 628.896,A -85,B 0,C 180,E1 -2253.868,E2 -2253.868} C_VEL
LIN {X 0,Y 572.963,Z 624.949,A -85,B 0,C 180,E1 -2254.925,E2 -2254.925} C_VEL
LIN {X 0,Y 573.064,Z 618.878,A -85,B 0,C 180,E1 -2256.16,E2 -2256.16} C_VEL
LIN {X 0,Y 573.119,Z 612.239,A -85,B 0,C 180,E1 -2257.221,E2 -2257.221} C_VEL
LIN {X 0,Y 573.201,Z 603.992,A -85,B 0,C 180,E1 -2258.283,E2 -2258.283} C_VEL
LIN {X 0,Y 573.286,Z 595.541,A -85,B 0,C 180,E1 -2259.17,E2 -2259.17} C_VEL
LIN {X 0,Y 573.423,Z 585.101,A -85,B 0,C 180,E1 -2260.058,E2 -2260.058} C_VEL
LIN {X 0,Y 573.528,Z 573.358,A -85,B 0,C 180,E1 -2260.858,E2 -2260.858} C_VEL
LIN {X 0,Y 573.652,Z 562.288,A -85,B 0,C 180,E1 -2261.447,E2 -2261.447} C_VEL
